(*
---Get axis errir txt
*)
METHOD Get_ErrTxt : STRING(255)
VAR_INPUT
END_VAR
Get_ErrTxt:=fb_motionModule.axisErrTxt;
END_METHOD

(*
---Get axis HOME condition
*)
METHOD Get_HomeCondition : BOOL
VAR_INPUT
END_VAR
Get_HomeCondition:=fb_motionModule.homeCondition;
END_METHOD

(*
---Get axis home state
*)
METHOD Get_HomeState : BOOL
VAR_INPUT
END_VAR
Get_HomeState:=fb_motionModule.axisHomeState;
END_METHOD

(*
---Get axis JOG condition
*)
METHOD Get_JogCondition : BOOL
VAR_INPUT
END_VAR
Get_JogCondition:=fb_motionModule.jogCondition;
END_METHOD

(*
---Get axis Modulo move condition
*)
METHOD Get_ModuloCondition : BOOL
VAR_INPUT
END_VAR
Get_ModuloCondition:=fb_motionModule.moveModuloCondition;
END_METHOD

(*
---Get axis pause state
*)
METHOD Get_Pause : BOOL
VAR_INPUT
END_VAR
Get_Pause:=fb_motionModule.axisPause;
END_METHOD

(*
---Get axis_ref pointer
*)
METHOD Get_pAXIS_REF : POINTER TO AXIS_REF
VAR_INPUT
END_VAR
Get_pAXIS_REF:=fb_motionModule.pAxis;
END_METHOD

(*
---Get axis REL condition
*)
METHOD Get_RelCondition : BOOL
VAR_INPUT
END_VAR
Get_RelCondition:=fb_motionModule.relCondition;
END_METHOD

(*
---Get axis SetPos condition
*)
METHOD Get_SetPosCondition : BOOL
VAR_INPUT
END_VAR
Get_SetPosCondition:=fb_motionModule.setCondition;
END_METHOD

(*
---Get axis VEL condition
*)
METHOD Get_VelCondition : BOOL
VAR_INPUT
END_VAR
Get_VelCondition:=fb_motionModule.velCondition;
END_METHOD

ACTION Obj_Instance:
fb_motionModule(
	axis:=axis,
	PLimitSwitch:= bPLimitSwitch, 
	NLimitSwitch:= bNLimitSwitch, 
	DOGPointSwitch:= bDOGPointSwitch, 
	bP_Pos:=bP_Pos,
	bN_Pos:=bN_Pos,
	torqueAlmValue:=bTorqueAlmValue,
	torqueEN:=bTorqueEN,
	motorType:= eMotorType, 
	moduloMode:= bModuloMode, 
	errorID:= nBaseErrID, 
	nameTXT:= sNameTXT, 
	axisEnable:= TRUE, 
	bE_Stop:= bE_Stop, 
	axisOverride:= , 
	//ctrlMode:= eCtrlMode,
	hmiEN:= hmiEN, 
	powerEnable:= , 
	powerEnable_Positive:= bEnablePositive, 
	powerEnable_Negative:= bEnableNegative, 
	enableSoftLimit:= bEnableSoftLimit, 
	softPLimitPos:= fSoftPLimitPos, 
	softNLimitPos:= fSoftNLimitPos, 
	axisStopFlag:= , 
	resetExecute:= , 
	pauseExecute:= , 
	jogExecute:= , 
	jogConditionOuter:= bJogConditionOuter, 
	jogDirection:= , 
	jogVelocity:= , 
	jogAcceleration:= , 
	jogDeceleration:= , 
	jogJerk:= , 
	stopExecute:= , 
	stopDeceleration:= , 
	stopJerk:= , 
	absExecute:= , 
	absMixedMovement:= , 
	absConditionOuter:= bAbsConditionOuter, 
	absPosition:= , 
	absVelocity:= , 
	absMixedPositionArray:= , 
	absMixedVelocityArray:= , 
	absMixedArrayLength:= , 
	absAcceleration:= , 
	absDeceleration:= , 
	absJerk:= , 
	relExecute:= , 
	relConditionOuter:= bRelConditionOuter, 
	relDistance:= , 
	relVelocity:= , 
	relAcceleration:= , 
	relDeceleration:= , 
	relJerk:= , 
	velExecute:= , 
	velConditionOuter:= bVelConditionOuter, 
	velDirection:= , 
	velVelocity:= , 
	velAcceleration:= , 
	velDeceleration:= , 
	velJerk:= , 
	homeExecute:= , 
	homeConditionOuter:= bHomeConditionOuter, 
	homeDirection:= bHomeDirection, 
	homeMode:= eHomeMode, 
	homeLimitSwitch_To_DOGDistance:= fHomeLimitSwitch_To_DOGDistance, 
	homeOnlyDOGDistance:= fHomeOnlyDOGDistance, 
	homeOnlyDOGMaxDistance:= fHomeOnlyDOGMaxDistance, 
	homePosition:= fHomePosition, 
	homeCheckRange:= fHomeCheckRange, 
	homeVel:= fHomeVel, 
	homeVelSlow:= fHomeVelSlow, 
	setPosExecute:= , 
	setConditionOuter:= bSetConditionOuter, 
	setPosPosition:= , 
	setPosOptions:= , 
	moveModuloExecute:= , 
	moveModuloConditionOuter:= bMoveModuloConditionOuter, 
	moveModuloPosition:= , 
	moveModuloVelocity:= , 
	moveModuloAcceleration:= , 
	moveModuloDeceleration:= , 
	moveModuloJerk:= , 
	moveModuloDirection:= , 
	axisActualPos=> , 
	axisActualVel=> , 
	axisPause=> , 
	axisBusy=> , 
	axisDone=> , 
	axisError=> , 
	axisErrId=> , 
	axisErrTxt=> , 
	axisHomeState=> , 
	pAxis=> , 
	jogCondition=> , 
	absCondition=> , 
	relCondition=> , 
	velCondition=> , 
	homeCondition=> , 
	setCondition=> , 
	moveModuloCondition=> );
END_ACTION

(*
---Set Acceleration\Deceleration\Jerk
*)
METHOD Set_AccDecJerk : BOOL
VAR_INPUT
	acc:LREAL;//target Acceleration
	dec:LREAL;//target Deceleration
	jerk:LREAL;//target Jerk
END_VAR
fb_motionModule.jogAcceleration:=acc;
fb_motionModule.jogDeceleration:=dec;
fb_motionModule.jogJerk:=jerk;

fb_motionModule.stopDeceleration:=dec;
fb_motionModule.stopJerk:=jerk;

fb_motionModule.absAcceleration:=acc;
fb_motionModule.absDeceleration:=dec;
fb_motionModule.absJerk:=jerk;

fb_motionModule.relAcceleration:=acc;
fb_motionModule.relDeceleration:=dec;
fb_motionModule.relJerk:=jerk;

fb_motionModule.velAcceleration:=acc;
fb_motionModule.velDeceleration:=dec;
fb_motionModule.velJerk:=jerk;

fb_motionModule.moveModuloAcceleration:=acc;
fb_motionModule.moveModuloDeceleration:=dec;
fb_motionModule.moveModuloJerk:=jerk;

Set_AccDecJerk:=TRUE;
END_METHOD

(*
---Set axis override
*)
METHOD Set_Override : BOOL
VAR_INPUT
	override:LREAL;//target axis override
END_VAR
fb_motionModule.axisOverride:=override;

Set_Override:=TRUE;
END_METHOD

(*
---Set Power Enable
*)
METHOD Set_Power : BOOL
VAR_INPUT
	enable:BOOL;
END_VAR
fb_motionModule.powerEnable:=enable;
END_METHOD

ACTION VersionLog:
(*
Version: V1.0.0.0
/-----------------------------------------------/
Version: V1.0.0.1
修改：修改电机模块使能触发方式(Add method Set_Power)
/-----------------------------------------------/
Version: V1.0.0.2
修改：增加中文报警输出
/-----------------------------------------------/
Version: V1.0.0.3
修改：增加中优化代码
/-----------------------------------------------/
Version: V1.0.0.4
更新时间: 2020/10/06
修改：配合轴模块更新
/-----------------------------------------------/
*)
END_ACTION

END_FUNCTION_BLOCK

// ---- POUs/BaseModule/ActionModule/motorModule/MotionModule.TcPOU
(*
--报错编号0: 无报错
--报错编号1: E_Stop!!!
--报错编号2: Soft Limit Error
--报错编号3: PLimit Switch Error
--报错编号4: NLimit Switch Error
--报错编号5: Origin sensor cannot be searched
--报错编号6: Go Home Failed
--报错编号7: Absolute Move Error
--报错编号8: JOG Move Error
--报错编号9: Modulo Move Error
--报错编号10: Relative Move Error
--报错编号11: Set Position Error
--报错编号12: Axis Stop Error
--报错编号13: Velocity Move Error
--报错编号14: mcPower Error
--报错编号15: mcReset Error
--报错编号16: axis_Status_Error
*)
FUNCTION_BLOCK MotionModule
VAR_IN_OUT
	axis							:AXIS_REF;//链接到实际的轴
END_VAR
VAR_INPUT
	HMIItf							:motionModuleDataHMI;//for manual and IO control//用于生成一个轴对象手动界面
	PLimitSwitch					:BOOL:=TRUE;//MC轴正限位感应信号
	NLimitSwitch					:BOOL:=TRUE;//MC轴负限位感应信号
	DOGPointSwitch					:BOOL:=FALSE;//MC轴原点感应信号
	bP_Pos							:LREAL:=0.777;	 //正向位置(开门）
	bN_Pos							:LREAL:=0.777;	 //负向位置(关门）

	motorType						:MotorType:=MotorType_Default;//设置电机的类型
	moduloMode						:BOOL:=FALSE;// modulo Mode, 旋转模式
	errorID							:UDINT:=0;//电机错误报警分配的起始ID
	nameTXT							:STRING(255):='';//电机名字

	axisEnable						:BOOL:=TRUE;//轴触摸屏是否启用
	bE_Stop							:BOOL:=TRUE;//急停信号
	axisOverride					:LREAL:=100.0;//轴运动的速度比
	//ctrlMode						:ControlMode:=ControlMode.eManualCtrMode;//eManualCtrMode or eAutoCtrMode
	hmiEN							:BOOL:=TRUE;//HMI 启用条件
	torqueEN						:BOOL:=FALSE;// 启用条件
	torqueAlmValue					:LREAL;// 报警扭力值
//POWER
	powerEnable						:BOOL:=TRUE;//轴使能触发
	powerEnable_Positive			:BOOL:=TRUE;//轴允许正转
	powerEnable_Negative			:BOOL:=TRUE;//轴允许反转
//Soft limit
	enableSoftLimit					:BOOL:=FALSE;//轴软限位 启用信号
	softPLimitPos					:LREAL:=9999999;//轴软限位 正向软限位
	softNLimitPos					:LREAL:=-9999999;//轴软限位 负向软限位
//STOP
	axisStopFlag					:BOOL:=FALSE;//轴是否停止
//RESET
	resetExecute					:BOOL:=TRUE;
	resetExecute2					:BOOL:=TRUE;//轴Reset的触发信号
//PAUSE
	pauseExecute					:BOOL:=FALSE;//轴Pause的触发信号
//JOG
	jogExecute						:BOOL:=FALSE;//轴JOG的触发信号
	jogConditionOuter				:BOOL:=TRUE;//轴JOG运动启停条件Outer
	jogDirection					:BOOL:=TRUE;//轴JOG运动方向信号, TRUE--正向，FALSE--反向
	jogVelocity						:LREAL:=10;//轴JOG运动运行速率值
	jogAcceleration					:LREAL:=0;//轴JOG运动加速度值
	jogDeceleration					:LREAL:=0;//轴JOG运动减速度值
	jogJerk							:LREAL:=0;//轴JOG运动 加加速度
//STOP
	stopExecute						:BOOL:=FALSE;//轴STOP的触发信号
	//20211029新增---by CPH 目的是仅有原点信号进行回零时，Stopexcute或者ACT——Stop动作无法似的该轴停止
	stoptemp						:BOOL:=FALSE;//轴STOP中转变量，主要传递给HMI界面的Stop指令
	stopDeceleration				:LREAL:=0;//轴STOP运动减速度值
	stopJerk						:LREAL:=0;//轴STOP运动 加加速度
//MoveAbsolute
	absExecute						:BOOL:=FALSE;//轴绝对运动的启停信号
	absMixedMovement				:BOOL:=FALSE;//轴绝对运动的混合变速运动 启用
	absConditionOuter				:BOOL:=TRUE;//轴绝对运动启停条件Outer
	absPosition						:LREAL:=0;//轴绝对运动 目标位置
	absVelocity						:LREAL:=0; //轴绝对运动 运行速率值
	absMixedPositionArray			:ARRAY [1..50] OF LREAL;//轴绝对运动 混合目标位置 变速触发位置数组 最大50个 数组最后一个位置为终点目标位置
	absMixedVelocityArray			:ARRAY [1..50] OF LREAL;//轴绝对运动 混合目标位置 变速触发位置数组 最大50个
	absMixedArrayLength				:UDINT:=0;//轴绝对运动 混合变速触发位置数组 长度 最大50个
	absAcceleration					:LREAL:=0;//轴绝对运动 加速度值
	absDeceleration					:LREAL:=0;//轴绝对运动 减速度值
	absJerk							:LREAL:=0;//轴绝对运动 加加速度
//Relative
	relExecute						:BOOL:=FALSE;//轴相对运动的启停信号
	relConditionOuter				:BOOL:=TRUE;//轴相对运动启停条件Outer
	relDistance						:LREAL:=0; //轴相对运动目标位置
	relVelocity						:LREAL:=0; //轴相对运动运行速率值
	relAcceleration					:LREAL:=0;//轴相对运动加速度值
	relDeceleration					:LREAL:=0;//轴相对运动减速度值
	relJerk							:LREAL:=0;//轴相对运动 加加速度
//Velocity
	velExecute						:BOOL:=FALSE;//轴速度模式运动的启停信号
	velConditionOuter				:BOOL:=TRUE;//轴速度模式启停条件Outer
	velDirection					:BOOL:=TRUE;//方向信号，TRUE--MC_Positive_Direction, FALSE--MC_Negative_Direction
	velVelocity						:LREAL:=10; //轴速度模式运行速率值
	velAcceleration					:LREAL:=0;//轴速度模式加速度值
	velDeceleration					:LREAL:=0;//轴速度模式减速度值
	velJerk							:LREAL:=0;//轴速度模式 加加速度
//Home
	homeExecute						:BOOL:=FALSE;//轴go home的启停信号
	homeConditionOuter				:BOOL:=TRUE;//轴go home的启停条件Outer
	homeDirection					:BOOL:=TRUE;//轴go home方向 TRUE--正方向，FALSE--负方向
	homeMode						:MotorHomeMode:=MotorHomeMode.MotorHomeMode_Default;//轴go home 模式
	homeLimitSwitch_To_DOGDistance	:LREAL:=5;//电机Home模式为 MotorHomeMode_PLimitSwitch_To_DOG/MotorHomeMode_NLimitSwitch_To_DOG 时, 脱离限位为原点的距离值
	homeOnlyDOGDistance				:LREAL:=5;//电机Home模式为 MotorHomeMode_OnlyDOGPointSwitch 时, 执行往复搜寻动作的幅度
	homeOnlyDOGMaxDistance			:LREAL:=360;//电机Home模式为 MotorHomeMode_OnlyDOGPointSwitch 时, 执行往复搜寻动作幅度的最大值
	homePosition					:LREAL:=0;
	homeCheckRange					:LREAL:=0.01;//轴go home执行完后当前位置判断值
	homeVel							:LREAL:=10;//轴go home 查找限位的速率
	homeVelSlow						:LREAL:=5;//轴go home 查找限位的爬行速率
//SetPositon
	setPosExecute					:BOOL:=FALSE;//轴当前位置设定启停信号
	setConditionOuter				:BOOL:=TRUE;//轴当前位置设定启停条件Outer
	setPosPosition					:LREAL:=0; //轴当前位置设定值
	setPosOptions					:ST_SetPositionOptions;//:=ST_SetPositionOptions.ClearPositionLag;
//MC_MoveModulo
	moveModuloExecute				:BOOL:=FALSE;//轴模运动的启停信号
	moveModuloConditionOuter		:BOOL:=TRUE;//轴模运动启停条件Outer
	moveModuloPosition				:LREAL:=0;//轴模运动目标位置
	moveModuloVelocity				:LREAL:=100; //轴模运动运行速率值
	moveModuloAcceleration			:LREAL:=0;//轴模运动加速度值
	moveModuloDeceleration			:LREAL:=0;//轴模运动减速度值
	moveModuloJerk					:LREAL:=0;//轴模运动 加加速度
	moveModuloDirection				:MC_Direction:=MC_Direction.MC_Shortest_Way;//MC_Shortest_Way; MC_Positive_Direction; MC_Negative_Direction
	noteWTXT_jog					:WSTRING(255):="";// 轴点动动作NoteTXT 中文
	noteWTXT_abs					:WSTRING(255):="";// 轴绝对定位动作NoteTXT 中文
	noteWTXT_rel					:WSTRING(255):="";// 轴相对定位动作NoteTXT 中文
	noteWTXT_vel					:WSTRING(255):="";// 轴速度运动动作NoteTXT 中文
END_VAR
VAR_OUTPUT
	axisActualPos					:LREAL:=0;//轴的实际位置
	axisActualVel					:LREAL:=0;//轴的实际速率
	axisActualtorque				:LREAL:=0;//轴的实际扭力
	axisPause						:BOOL;//轴的Pause状态
	axisBusy						:BOOL;//轴的Busy状态
	axisDone						:BOOL;//轴的Done状态
	axisError						:BOOL;//轴的Error状态
	axisErrId						:UDINT;//轴的Error Id值
	axisErrTxt						:STRING(255);//轴的报错文本信息
	axisErrWTxt						:WSTRING(255);//轴的报错文本信息 中文
	axisHomeState					:BOOL:=FALSE;//轴的原点状态
	pAxis	  						:POINTER TO AXIS_REF;
	
	note_jog						:BOOL:=FALSE;// 点动条件不满足
	jogCondition					:BOOL;//轴JOG运动启动条件
	note_abs						:BOOL:=FALSE;// 绝对定位条件不满足
	absCondition					:BOOL;//轴绝对运动启动条件
	note_rel						:BOOL:=FALSE;// 相对定位条件不满足
	relCondition					:BOOL;//轴相对运动启动条件
	note_vel						:BOOL:=FALSE;// 速度条件不满足
	velCondition					:BOOL;//轴速度模式启动条件
	note_home						:BOOL:=FALSE;// 回原条件不满足
	homeCondition					:BOOL;//轴go home的启动条件
	setCondition					:BOOL;//轴当前位置设定启动条件
	moveModuloCondition				:BOOL;//轴模运动启动条件
END_VAR
VAR
	//axis							:AXIS_REF;//链接到实际的轴

	op_mode 				AT%Q*	:SINT:=8;//RxPDO1的Modes of operation---只用于横川DD马达(高创驱动器)
	mode_display 			AT%I*	:SINT;//TxPDO1的Modes of operation display---只用于横川DD马达(高创驱动器)
	maxProfileVelocity  	AT%Q*	:UDINT:=838860800 ; //链接到伺服的Maxprofilevelocity
	statusWord 				AT%I*	:UINT; //链接到伺服的Statusword
	
	torqueAlmErr					:BOOL;// 报警扭力
	torqueErr_Rtrig					:R_TRIG;
	bInit							:BOOL:=FALSE;
	mcBusy							:BOOL;
	mcError							:BOOL;
	mcPower							:MC_Power;
	mcReset							:MC_Reset;
	mcStop							:MC_Stop;
//	mcHalt							:MC_Halt;
	mcJog							:MC_Jog;
	mcABSMove						:MC_MoveAbsolute;
	mcABSMove2						:MC_MoveAbsolute;
	mcABSMove3						:MC_MoveAbsolute;
	mcABSMove4						:MC_MoveAbsolute;
	absBufferMode					:MC_BufferMode:=MC_BufferMode.MC_Aborting;
	mcRel							:MC_MoveRelative;
	mcVel							:MC_MoveVelocity;
	mcHome							:MC_Home;
	mcSetPos						:MC_SetPosition;
	mcMoveModulo					:MC_MoveModulo;
//STOP
	stopBusy						:BOOL;
	stopDone						:BOOL;
	stopErrorDone					:BOOL;
	stopTrigR1						:R_Trig;//上升沿触发
	stopStep						:UINT:=0;
	stopTimeout						:TON;
//Jog
	jogBusy							:BOOL;
	jogDone							:BOOL;
	jogErrorDone					:BOOL;
	jogForward						:BOOL:=FALSE;//轴JOG运动正向启停信号
	jogBackwards					:BOOL:=FALSE;//轴JOG运动反向启停信号
	jogTrigR1						:R_Trig;//上升沿触发
	jogTrigF1						:F_Trig;//上升沿触发
	jogTrigR1_NAiko					:R_Trig;//上升沿触发
	jogTrigF1_NAiko					:F_Trig;//上升沿触发
	jogTrigR1_PAiko					:R_Trig;//上升沿触发
	jogTrigF1_PAiko					:F_Trig;//上升沿触发
	
	jogStep							:UINT:=0;
//Absolute
	absBusy							:BOOL;
	absDone							:BOOL;
	absErrorDone					:BOOL;
	absTrigR1						:R_Trig;//上升沿触发
	absT1							:TON;//长按计时
	absRP							:R_TRIG;// 短按执行去开门位置
	absRN							:R_TRIG;// 短按执行去关门位置
	absStep							:UINT:=0;
	absMixedCount					:UDINT:=0;
//Relative
	relBusy							:BOOL;
	relDone							:BOOL;
	relErrorDone					:BOOL;
	relTrigR1						:R_Trig;//上升沿触发
	relT1							:TON;//长按计时
	relStep							:UINT:=0;
//Velocity 
	velBusy							:BOOL;
	velDone							:BOOL;
	velErrorDone					:BOOL;
	velTrigR1						:R_Trig;//上升沿触发
	velStep							:UINT:=0;
	velChangeVel					:BOOL:=FALSE;//轴速度模式运动 速度改变触发
	
	velTrigR1_NAiko					:R_Trig;//上升沿触发
	velTrigF1_NAiko					:F_Trig;//上升沿触发
	velTrigR1_PAiko					:R_Trig;//上升沿触发
	velTrigF1_PAiko					:F_Trig;//上升沿触发
//Home
	goHomeTrigR1					:R_Trig;//上升沿触发
	goHomeTrigF1					:F_Trig;//下降沿检测
	goHomeDelayTon					:Ton;
	goHomeDelayTime					:TIME:=T#100MS;
	goHomeRelDistance				:LREAL:=0; //Home 轴相对运动目标位置
	goHomeRelVelocity				:LREAL:=0; //Home 轴相对运动运行速率值

	homeDone						:BOOL;
	homeErrorDone					:BOOL;
	homeBusy						:BOOL;
	homeStep						:UINT:=0;
//SetPositon
	setPosBusy						:BOOL;
	setPosDone						:BOOL;
	setPosErrorDone					:BOOL;
	setPosTrigR1					:R_Trig;//上升沿触发
	setPosStep						:UINT:=0;
//MC_MoveModulo
	moveModuloBusy					:BOOL;
	moveModuloDone					:BOOL;
	moveModuloErrorDone				:BOOL;
	moveModuloStep					:UINT:=0;
//power
	powerTrigF1						:F_Trig;//下降沿触发
	powerEnable_Inner				:BOOL:=TRUE;//轴使能触发 内部的
	powerReady						:BOOL;
//reset
	resetBusy						:BOOL;
	resetDone						:BOOL;
	resetErrorDone					:BOOL;
	resetTrigR1						:R_Trig;//上升沿触发
	resetTrigR2						:R_Trig;//上升沿触发
	resetStep						:UINT:=0;
//pause
	pause_Manual_F_Trig				:F_Trig;//HMI暂停 上升沿触发
	pauseR_Trig						:R_Trig;//暂停 上升沿触发
	pauseF_Trig						:F_Trig;//暂停 下降沿触发
//Loop
	loopRelGoTrigR1					:R_Trig;//上升沿触发
	loopAbsGoTrigR1					:R_Trig;//上升沿触发
	loopRelGoT1						:TON;//长按计时
	loopAbsGoT1						:TON;//长按计时
	loopStepHome					:UINT:=0;
	loopStep						:UINT:=0;
	loopRelGo						:BOOL:=FALSE;//loop 相对运动启动
	loopGoHome						:BOOL:=FALSE;//loop 相对运动启动 回原方式
	loopAbsGo						:BOOL:=FALSE;//loop 绝对运动启动
	loopFirstPoint					:LREAL:=0;//loop 第1个点
	loopSecondPoint					:LREAL:=0;//loop 第2个点
	loopGoVel						:LREAL:=10;//loop 运动速率
	loopCycle						:UINT:=0;//loop 循环次数 一次往复才算一次
	loopCycleMax					:UINT:=0;//loop 循环次数 一次往复才算一次
	loopWatingTime					:UINT:=1000;//loop 停留时间（单位ms）
	loopCycleTimes					:UINT:=0;//loop 循环次数 一次往复才算一次
	loopCycleTimesHome				:UINT:=0;//loop 循环次数 一次往复才算一次
	loopWatingTON					:TON;
//Other
	bPLimitSwitch					:BOOL:=TRUE;//MC轴正限位感应信号
	bNLimitSwitch					:BOOL:=TRUE;//MC轴负限位感应信号
	bSoftPLimit						:BOOL:=TRUE;//
	bSoftNLimit						:BOOL:=TRUE;//
	
	overrideSet						:LREAL:=100.0;//轴运动的速度比 设置
	overrideTemp					:LREAL:=100.0;//轴运动的速度比 缓存
	stopTon							:TON;
	manualStep						:UINT:=0;
	busy							:BOOL:=FALSE;
	busyR_Trig						:R_Trig;
	doneR_Trig						:R_Trig;
	motorError						:BOOL:=FALSE;
	PTPErrID						:UDINT;
	errorStep						:UINT:=0;
	
	//OnlyDOG Go home TON
	t1Temp							:TON;
	//Home Delay
	tHomeTemp						:TON;
	loopHomeToPosGoT1				:TON;//长按计时
	loopHomeToPosTrigR1				:R_Trig;//上升沿触发
	noteTON_P:tON;            // 操作提示标志位延时继电器
	noteTON_N:tON;            // 操作提示标志位延时继电器
	noteRTrig_P:R_TRIG;          // 操作提示
	noteRTrig_N:R_TRIG;          // 操作提示
END_VAR

(*
Please refer to the VersionLog file for version records
*)
axis.ReadStatus();
IF moduloMode THEN
	axisActualPos:=axis.NcToPlc.ModuloActPos;//获取轴的实际位置, modulo Mode
ELSE
	axisActualPos:=axis.NcToPlc.ActPos;//获取轴的实际位置
END_IF
axisActualtorque:=axis.NcToPlc.ActTorque;
IF torqueEN THEN// 扭力报警监控
	IF ABS(axisActualtorque)>torqueAlmValue THEN
		torqueAlmErr:=TRUE;
	ELSE
		torqueAlmErr:=FALSE;
	END_IF
ELSE
	torqueAlmErr:=FALSE;
END_IF
torqueErr_Rtrig(CLK:=torqueAlmErr);
IF torqueErr_Rtrig.Q THEN
	errorStep:=17;
END_IF
axisActualVel:=axis.NcToPlc.ActVelo;//获取轴的实际速率
pAxis:=ADR(axis);
powerReady:=mcPower.Status;

IF NOT bE_Stop THEN
	axisStopFlag:=TRUE;
	axisHomeState:=FALSE;
	homeBusy:=FALSE;
	errorStep:=1;
END_IF
bPLimitSwitch:=PLimitSwitch;
bNLimitSwitch:=NLimitSwitch;
bSoftPLimit:=(NOT enableSoftLimit OR ((enableSoftLimit AND axisActualPos<softPLimitPos) OR homeBusy));
bSoftNLimit:=(NOT enableSoftLimit OR ((enableSoftLimit AND axisActualPos>softNLimitPos) OR homeBusy));

busy:=stopBusy OR jogBusy OR absBusy OR relBusy OR velBusy (*OR homeBusy*) OR 0<>loopStep;
mcBusy:=mcStop.Busy OR mcJog.Busy OR mcABSMove.Busy OR mcABSMove2.Busy 
			OR mcABSMove3.Busy OR mcABSMove4.Busy OR mcRel.Busy 
			OR mcVel.Busy OR mcHome.Busy OR mcSetPos.Busy OR mcMoveModulo.Busy;
axisBusy:=(mcBusy OR busy OR homeBusy OR (0<>axis.NcToPlc.AxisState));
busyR_Trig(CLK:=axisBusy);
IF busyR_Trig.Q THEN
	jogDone:=FALSE;
	absDone:=FALSE;
	relDone:=FALSE;
	velDone:=FALSE;
	homeDone:=FALSE;
	setPosDone:=FALSE;
	stopDone:=FALSE;
	moveModuloDone:=FALSE;
	
	axisDone:=FALSE;
END_IF

doneR_Trig(CLK:=(jogDone OR absDone OR relDone OR velDone OR homeDone OR setPosDone (*OR stopDone*) OR moveModuloDone) AND NOT axisBusy);
IF doneR_Trig.Q THEN
	axisDone:=TRUE;
	
	jogDone:=FALSE;
	absDone:=FALSE;
	relDone:=FALSE;
	velDone:=FALSE;
	homeDone:=FALSE;
	setPosDone:=FALSE;
	stopDone:=FALSE;
	moveModuloDone:=FALSE;
END_IF

IF axis.Status.Error OR 0<>axis.NcToPlc.ErrorCode THEN
	errorStep:=16;
END_IF
Error_ACT();
mcError:=mcPower.Error OR mcReset.Error OR mcStop.Error OR mcJog.Error OR mcABSMove.Error 
			OR mcABSMove2.Error OR mcABSMove3.Error OR mcABSMove4.Error 
			 OR mcRel.Error OR mcVel.Error OR mcHome.Error OR mcSetPos.Error
			 OR mcMoveModulo.Error;
axisError:=(mcError OR axis.Status.Error OR 0<>axis.NcToPlc.ErrorCode OR NOT bE_Stop OR motorError OR torqueAlmErr);
Error_ACT();

IF NOT axisError THEN
	errorStep:=0;
END_IF

Power_ACT();
Reset_ACT();
ResetEx_ACT();
SetPause_ACT();
InitHMI_ACT();
ManualCtr_ACT();

Stop_ACT();
JogMove_ACT();
VelMove_ACT();
GoHome_ACT();
RelMove_ACT();
AbsMove_ACT();
MoveModulo_ACT();
SetPosition_ACT();
LoopMove_ACT();
LoopHomeToPos_ACT();
IF NOT bInit THEN
	bInit:=TRUE;
END_IF

busy:=stopBusy OR jogBusy OR absBusy OR relBusy OR velBusy (*OR homeBusy*) OR 0<>loopStep;
mcBusy:=mcStop.Busy OR mcJog.Busy OR mcABSMove.Busy OR mcABSMove2.Busy 
			OR mcABSMove3.Busy OR mcABSMove4.Busy OR mcRel.Busy 
			OR mcVel.Busy OR mcHome.Busy OR mcSetPos.Busy OR mcMoveModulo.Busy;
axisBusy:=(mcBusy OR busy OR homeBusy OR (0<>axis.NcToPlc.AxisState));
busyR_Trig(CLK:=axisBusy);
IF busyR_Trig.Q THEN
	jogDone:=FALSE;
	absDone:=FALSE;
	relDone:=FALSE;
	velDone:=FALSE;
	homeDone:=FALSE;
	setPosDone:=FALSE;
	stopDone:=FALSE;
	moveModuloDone:=FALSE;
	
	axisDone:=FALSE;
END_IF

doneR_Trig(CLK:=(jogDone OR absDone OR relDone OR velDone OR homeDone OR setPosDone (*OR stopDone*) OR moveModuloDone) AND NOT axisBusy);
IF doneR_Trig.Q THEN
	axisDone:=TRUE;
	
	jogDone:=FALSE;
	absDone:=FALSE;
	relDone:=FALSE;
	velDone:=FALSE;
	homeDone:=FALSE;
	setPosDone:=FALSE;
	stopDone:=FALSE;
	moveModuloDone:=FALSE;
END_IF

ACTION AbsMove_ACT:
//轴绝对运动运行控制--absExecute触发条件是复归型
IF NOT bE_Stop THEN
	absStep:=0;
	absExecute:=FALSE;
END_IF
absCondition:=(axisHomeState AND NOT axisError 
				AND NOT axisStopFlag AND (NOT axisBusy OR 0<>loopStep) 
				AND powerReady AND absConditionOuter 
				AND bE_Stop AND NOT axisPause);

mcABSMove(
	Axis:=axis , 
	Execute:= , 
	Position:= , 
	Velocity:= , 
	Acceleration:= , 
	Deceleration:= , 
	Jerk:= , 
	BufferMode:= , 
	Options:= , 
	Done=> , 
	Busy=> , 
	Active=> , 
	CommandAborted=> , 
	Error=> , 
	ErrorID=> );
mcABSMove2(
	Axis:=axis , 
	Execute:= , 
	Position:= , 
	Velocity:= , 
	Acceleration:= , 
	Deceleration:= , 
	Jerk:= , 
	BufferMode:= , 
	Options:= , 
	Done=> , 
	Busy=> , 
	Active=> , 
	CommandAborted=> , 
	Error=> , 
	ErrorID=> );
mcABSMove3(
	Axis:=axis , 
	Execute:= , 
	Position:= , 
	Velocity:= , 
	Acceleration:= , 
	Deceleration:= , 
	Jerk:= , 
	BufferMode:= absBufferMode, 
	Options:= , 
	Done=> , 
	Busy=> , 
	Active=> , 
	CommandAborted=> , 
	Error=> , 
	ErrorID=> );
mcABSMove4(
	Axis:=axis , 
	Execute:= , 
	Position:= , 
	Velocity:= , 
	Acceleration:= , 
	Deceleration:= , 
	Jerk:= , 
	BufferMode:= absBufferMode, 
	Options:= , 
	Done=> , 
	Busy=> , 
	Active=> , 
	CommandAborted=> , 
	Error=> , 
	ErrorID=> );

CASE absStep OF
0:
	absBusy:=FALSE;
	IF absExecute AND (NOT absCondition OR NOT powerEnable_Negative OR NOT powerEnable_Positive OR absVelocity>0.2) THEN
		note_abs:=TRUE;
		note_jog:=FALSE;
		note_vel:=FALSE;
		note_home:=FALSE;
		note_rel:=FALSE;
	END_IF
	IF absExecute AND absCondition THEN
		absBusy:=TRUE;
		absDone:=FALSE;
		absErrorDone:=FALSE;
		note_abs:=FALSE;
		note_jog:=FALSE;
		note_vel:=FALSE;
		note_home:=FALSE;
		note_rel:=FALSE;
		IF NOT absMixedMovement THEN
			absStep:=20;//点到点运动
		ELSE
			absPosition:=absMixedPositionArray[absMixedArrayLength];
			absStep:=100;//多段变速运动
		END_IF
	END_IF
	absExecute:=FALSE;
	absMixedMovement:=FALSE;
	absMixedCount:=1;
	mcABSMove(
		Axis:=axis , 
		Execute:=FALSE ,);
	mcABSMove2(
		Axis:=axis , 
		Execute:=FALSE ,);
	mcABSMove3(
		Axis:=axis , 
		Execute:=FALSE ,);
	mcABSMove4(
		Axis:=axis , 
		Execute:=FALSE ,);
20:
//	正确逻辑
	IF NOT bPLimitSwitch OR NOT bNLimitSwitch OR NOT bSoftPLimit OR NOT bSoftNLimit OR NOT powerEnable_Positive OR NOT powerEnable_Negative THEN
		axisStopFlag:=TRUE;

		IF NOT bPLimitSwitch THEN
			errorStep:=3;
		ELSIF NOT bNLimitSwitch THEN
			errorStep:=4;
		END_IF
		IF NOT bSoftPLimit OR NOT bSoftNLimit THEN
			errorStep:=2;
		END_IF
		IF NOT powerEnable_Positive OR NOT powerEnable_Negative THEN
			errorStep:=19;
		END_IF
		absStep:=10000;//error
		RETURN;
	END_IF
//	测试逻辑
//	IF NOT bSoftPLimit OR NOT bSoftNLimit THEN
//		axisStopFlag:=TRUE;

//		IF NOT bSoftPLimit OR NOT bSoftNLimit THEN
//			errorStep:=2;
//		END_IF
//		absStep:=10000;//error
//		RETURN;
//	END_IF
//	IF NOT bPLimitSwitch OR NOT bNLimitSwitch THEN
//		IF NOT bPLimitSwitch AND ABS(axisActualPos-absPosition)>6 THEN
//			axisStopFlag:=TRUE;
//			errorStep:=3;
//			absStep:=10000;//error
//			RETURN;
//		ELSIF NOT bNLimitSwitch AND ABS(axisActualPos-absPosition)>6 THEN
//			axisStopFlag:=TRUE;
//			errorStep:=4;
//			absStep:=10000;//error
//			RETURN;
//		END_IF
//	END_IF
	mcABSMove(
		Axis:=axis , 
		Execute:=TRUE , 
		Position:=absPosition , 
		Velocity:=absVelocity , 
		Acceleration:=absAcceleration , 
		Deceleration:=absDeceleration , 
		Jerk:=absJerk , 
		BufferMode:= , 
		Options:= , 
		Done=> , 
		Busy=> , 
		Active=> , 
		CommandAborted=> , 
		Error=> , 
		ErrorID=> );
// 正常
	IF mcABSMove.Done THEN//mcABSMove.Done信号只保持一个扫描周期
		absStep:=5000;//done
	ELSIF mcABSMove.Error OR mcABSMove.ErrorID<>0 THEN
		errorStep:=7;
		absStep:=10000;//error
	END_IF
// 测试逻辑
//	IF mcABSMove.Done THEN//mcABSMove.Done信号只保持一个扫描周期
//		IF NOT bSoftPLimit OR NOT bSoftNLimit THEN
//			absStep:=5000;//done
//		ELSE
//			errorStep:=7;
//			absStep:=10000;//error
//		END_IF
//	ELSIF mcABSMove.Error OR mcABSMove.ErrorID<>0 THEN
//		errorStep:=7;
//		absStep:=10000;//error
//	END_IF

	IF axisStopFlag OR NOT powerReady OR 0<>stopStep THEN
		absStep:=4000;//stop
	END_IF

//变速运动
100:
	IF NOT bPLimitSwitch OR NOT bNLimitSwitch OR NOT bSoftPLimit OR NOT bSoftNLimit OR NOT powerEnable_Positive OR NOT powerEnable_Negative THEN
		axisStopFlag:=TRUE;

		IF NOT bPLimitSwitch THEN
			errorStep:=3;
		ELSIF NOT bNLimitSwitch THEN
			errorStep:=4;
		END_IF
		IF NOT bSoftPLimit OR NOT bSoftNLimit THEN
			errorStep:=2;
		END_IF
		IF NOT powerEnable_Positive OR NOT powerEnable_Negative THEN
			errorStep:=19;
		END_IF
		absStep:=10000;//error
		RETURN;
	END_IF
	mcABSMove2(
		Axis:=axis , 
		Execute:=TRUE , 
		Position:=absMixedPositionArray[absMixedCount] , 
		Velocity:=absMixedVelocityArray[absMixedCount] , 
		Acceleration:=absAcceleration , 
		Deceleration:=absDeceleration , 
		Jerk:=absJerk , 
		BufferMode:= , 
		Options:= , 
		Done=> , 
		Busy=> , 
		Active=> , 
		CommandAborted=> , 
		Error=> , 
		ErrorID=> );
	
	IF mcABSMove2.Busy AND (absMixedCount<absMixedArrayLength) THEN
		mcABSMove3(
			Axis:=axis , 
			Execute:=FALSE ,);
		IF absMixedVelocityArray[absMixedCount]>absMixedVelocityArray[absMixedCount+1] THEN
			absBufferMode:=MC_BufferMode.MC_BlendingNext;
		ELSE
			absBufferMode:=MC_BufferMode.MC_BlendingPrevious;
		END_IF
		absMixedCount:=absMixedCount+1;
		absStep:=110;
	END_IF
	IF mcABSMove2.Done THEN//mcABSMove.Done信号只保持一个扫描周期
		absStep:=5000;//done
	ELSIF mcABSMove2.Error OR mcABSMove2.ErrorID<>0 THEN
		errorStep:=7;
		absStep:=10000;//error
	END_IF

	IF axisStopFlag OR NOT powerReady OR 0<>stopStep THEN
		absStep:=4000;//stop
	END_IF
110:
	IF NOT bPLimitSwitch OR NOT bNLimitSwitch OR NOT bSoftPLimit OR NOT bSoftNLimit OR NOT powerEnable_Positive OR NOT powerEnable_Negative THEN
		axisStopFlag:=TRUE;

		IF NOT bPLimitSwitch THEN
			errorStep:=3;
		ELSIF NOT bNLimitSwitch THEN
			errorStep:=4;
		END_IF
		IF NOT bSoftPLimit OR NOT bSoftNLimit THEN
			errorStep:=2;
		END_IF
		IF NOT powerEnable_Positive OR NOT powerEnable_Negative THEN
			errorStep:=19;
		END_IF
		absStep:=10000;//error
		RETURN;
	END_IF
	mcABSMove3(
		Axis:=axis , 
		Execute:=TRUE , 
		Position:=absMixedPositionArray[absMixedCount] , 
		Velocity:=absMixedVelocityArray[absMixedCount] , 
		Acceleration:=absAcceleration , 
		Deceleration:=absDeceleration , 
		Jerk:=absJerk , 
		BufferMode:= , 
		Options:= , 
		Done=> , 
		Busy=> , 
		Active=> , 
		CommandAborted=> , 
		Error=> , 
		ErrorID=> );
	
	IF mcABSMove3.Busy AND NOT mcABSMove2.Busy AND NOT mcABSMove4.Busy AND (absMixedCount<absMixedArrayLength) THEN
		mcABSMove4(
			Axis:=axis , 
			Execute:=FALSE ,);
		IF absMixedVelocityArray[absMixedCount]>absMixedVelocityArray[absMixedCount+1] THEN
			absBufferMode:=MC_BufferMode.MC_BlendingNext;
		ELSE
			absBufferMode:=MC_BufferMode.MC_BlendingPrevious;
		END_IF
		absMixedCount:=absMixedCount+1;
		absStep:=120;
	END_IF
	IF mcABSMove3.Done THEN//mcABSMove.Done信号只保持一个扫描周期
		absStep:=5000;//done
	ELSIF mcABSMove3.Error OR mcABSMove3.ErrorID<>0 THEN
		errorStep:=7;
		absStep:=10000;//error
	END_IF

	IF axisStopFlag OR NOT powerReady OR 0<>stopStep THEN
		absStep:=4000;//stop
	END_IF
120:
	IF NOT bPLimitSwitch OR NOT bNLimitSwitch OR NOT bSoftPLimit OR NOT bSoftNLimit OR NOT powerEnable_Positive OR NOT powerEnable_Negative THEN
		axisStopFlag:=TRUE;

		IF NOT bPLimitSwitch THEN
			errorStep:=3;
		ELSIF NOT bNLimitSwitch THEN
			errorStep:=4;
		END_IF
		IF NOT bSoftPLimit OR NOT bSoftNLimit THEN
			errorStep:=2;
		END_IF
		IF NOT powerEnable_Positive OR NOT powerEnable_Negative THEN
			errorStep:=19;
		END_IF
		absStep:=10000;//error
		RETURN;
	END_IF
	mcABSMove4(
		Axis:=axis , 
		Execute:=TRUE , 
		Position:=absMixedPositionArray[absMixedCount] , 
		Velocity:=absMixedVelocityArray[absMixedCount] , 
		Acceleration:=absAcceleration , 
		Deceleration:=absDeceleration , 
		Jerk:=absJerk , 
		BufferMode:= , 
		Options:= , 
		Done=> , 
		Busy=> , 
		Active=> , 
		CommandAborted=> , 
		Error=> , 
		ErrorID=> );
	
	IF mcABSMove4.Busy AND NOT mcABSMove3.Busy AND (absMixedCount<absMixedArrayLength) THEN
		mcABSMove3(
			Axis:=axis , 
			Execute:=FALSE ,);
		IF absMixedVelocityArray[absMixedCount]>absMixedVelocityArray[absMixedCount+1] THEN
			absBufferMode:=MC_BufferMode.MC_BlendingNext;
		ELSE
			absBufferMode:=MC_BufferMode.MC_BlendingPrevious;
		END_IF
		absMixedCount:=absMixedCount+1;
		absStep:=110;
	END_IF
	IF mcABSMove4.Done THEN//mcABSMove.Done信号只保持一个扫描周期
		absStep:=5000;//done
	ELSIF mcABSMove4.Error OR mcABSMove4.ErrorID<>0 THEN
		errorStep:=7;
		absStep:=10000;//error
	END_IF

	IF axisStopFlag OR NOT powerReady OR 0<>stopStep THEN
		absStep:=4000;//stop
	END_IF
	
4000://Stop
	mcABSMove(
		Axis:=axis , 
		Execute:=FALSE ,);
	mcABSMove2(
		Axis:=axis , 
		Execute:=FALSE ,);
	mcABSMove3(
		Axis:=axis , 
		Execute:=FALSE ,);
	mcABSMove4(
		Axis:=axis , 
		Execute:=FALSE ,);
	absExecute:=FALSE;
	absBusy:=FALSE;
	absDone:=FALSE;
	absErrorDone:=FALSE;
	absStep:=0;
5000://Done
	mcABSMove(
		Axis:=axis , 
		Execute:=FALSE ,);
	mcABSMove2(
		Axis:=axis , 
		Execute:=FALSE ,);
	mcABSMove3(
		Axis:=axis , 
		Execute:=FALSE ,);
	mcABSMove4(
		Axis:=axis , 
		Execute:=FALSE ,);
	absExecute:=FALSE;
	absBusy:=FALSE;
	absDone:=TRUE;
	absErrorDone:=FALSE;
	absStep:=0;
10000://Error
	mcABSMove(
		Axis:=axis , 
		Execute:=FALSE ,);
	mcABSMove2(
		Axis:=axis , 
		Execute:=FALSE ,);
	mcABSMove3(
		Axis:=axis , 
		Execute:=FALSE ,);
	mcABSMove4(
		Axis:=axis , 
		Execute:=FALSE ,);
	absExecute:=FALSE;
	absBusy:=FALSE;
	absDone:=FALSE;
	absErrorDone:=TRUE;
	absStep:=0;
END_CASE
END_ACTION

//设定速度运行模式的方向和速度
METHOD changeVelVel
VAR_INPUT
	vel:LREAL;//速度设定
END_VAR
velChangeVel:=TRUE;
velVelocity:=vel;
END_METHOD

ACTION Error_ACT:
CASE errorStep OF
	0:
		motorError:=FALSE;
		axisErrId:=0;
		axisErrTxt:='';
		axisErrWTxt:="";
		PTPErrID:=0;
 (*
	1:
		motorError:=TRUE;
		axisErrId:=errorID+errorStep;
		axisErrTxt:=CONCAT(STR1:=nameTXT,STR2:=' E_Stop!!!');
		axisErrWTxt:=WCONCAT(STR1:=TO_WSTRING(nameTXT),STR2:=" 急停错误!!!");
	2:
		motorError:=TRUE;
		axisErrId:=errorID+errorStep;
		axisErrTxt:=CONCAT(STR1:=nameTXT,STR2:=' Soft Limit Error');
		axisErrWTxt:=WCONCAT(STR1:=TO_WSTRING(nameTXT),STR2:=" 软限位错误");
	3:
		motorError:=TRUE;
		axisErrId:=errorID+errorStep;
		axisErrTxt:=CONCAT(STR1:=nameTXT,STR2:=' PLimit Switch Error');
		axisErrWTxt:=WCONCAT(STR1:=TO_WSTRING(nameTXT),STR2:=" 正限位感应错误");
	4:
		motorError:=TRUE;
		axisErrId:=errorID+errorStep;
		axisErrTxt:=CONCAT(STR1:=nameTXT,STR2:=' NLimit Switch Error');
		axisErrWTxt:=WCONCAT(STR1:=TO_WSTRING(nameTXT),STR2:=" 负限位感应错误");
	5:
		motorError:=TRUE;
		axisErrId:=errorID+errorStep;
		axisErrTxt:=CONCAT(STR1:=nameTXT,STR2:=' Origin sensor cannot be searched');
		axisErrWTxt:=WCONCAT(STR1:=TO_WSTRING(nameTXT),STR2:=" 原点信号无法被搜索到");
	6:
		motorError:=TRUE;
		axisErrId:=errorID+errorStep;
		axisErrTxt:=CONCAT(STR1:=nameTXT,STR2:=' Go Home Failed');
		axisErrWTxt:=WCONCAT(STR1:=TO_WSTRING(nameTXT),STR2:=" 回原点失败");
	7:
		motorError:=TRUE;
		axisErrId:=errorID+errorStep;
		axisErrTxt:=CONCAT(STR1:=nameTXT,STR2:=' Absolute Move Error');
		axisErrWTxt:=WCONCAT(STR1:=TO_WSTRING(nameTXT),STR2:=" 绝对定位错误");
	8:
		motorError:=TRUE;
		axisErrId:=errorID+errorStep;
		axisErrTxt:=CONCAT(STR1:=nameTXT,STR2:=' JOG Move Error');
		axisErrWTxt:=WCONCAT(STR1:=TO_WSTRING(nameTXT),STR2:=" JOG运动错误");
	9:
		motorError:=TRUE;
		axisErrId:=errorID+errorStep;
		axisErrTxt:=CONCAT(STR1:=nameTXT,STR2:=' Modulo Move Error');
		axisErrWTxt:=WCONCAT(STR1:=TO_WSTRING(nameTXT),STR2:=" 模值定位错误");
	10:
		motorError:=TRUE;
		axisErrId:=errorID+errorStep;
		axisErrTxt:=CONCAT(STR1:=nameTXT,STR2:=' Relative Move Error');
		axisErrWTxt:=WCONCAT(STR1:=TO_WSTRING(nameTXT),STR2:=" 相对定位错误");
	11:
		motorError:=TRUE;
		axisErrId:=errorID+errorStep;
		axisErrTxt:=CONCAT(STR1:=nameTXT,STR2:=' Set Position Error');
		axisErrWTxt:=WCONCAT(STR1:=TO_WSTRING(nameTXT),STR2:=" 设置位置错误");
	12:
		motorError:=TRUE;
		axisErrId:=errorID+errorStep;
		axisErrTxt:=CONCAT(STR1:=nameTXT,STR2:=' Axis Stop Error');
		axisErrWTxt:=WCONCAT(STR1:=TO_WSTRING(nameTXT),STR2:=" 轴停止错误");
	13:
		motorError:=TRUE;
		axisErrId:=errorID+errorStep;
		axisErrTxt:=CONCAT(STR1:=nameTXT,STR2:=' Velocity Move Error');
		axisErrWTxt:=WCONCAT(STR1:=TO_WSTRING(nameTXT),STR2:=" 速度运行错误");
	14:
		motorError:=TRUE;
		axisErrId:=errorID+errorStep;
		axisErrTxt:=CONCAT(STR1:=nameTXT,STR2:=' mcPower Error');
		axisErrWTxt:=WCONCAT(STR1:=TO_WSTRING(nameTXT),STR2:=" mcPower轴使能错误");
	15:
		motorError:=TRUE;
		axisErrId:=errorID+errorStep;
		axisErrTxt:=CONCAT(STR1:=nameTXT,STR2:=' mcReset Error');
		axisErrWTxt:=WCONCAT(STR1:=TO_WSTRING(nameTXT),STR2:=" mcReset轴复位错误");
	16:
		motorError:=TRUE;
		axisErrId:=errorID+errorStep;
		axisErrTxt:=CONCAT(STR1:=nameTXT,STR2:=' axis_Status_Error');
		axisErrWTxt:=WCONCAT(STR1:=TO_WSTRING(nameTXT),STR2:=" 轴状态错误");
 *)
	1..19:
		motorError:=TRUE;
		axisErrId:=getErrID(errorStep);
		axisErrTxt:=getErrTXT(errorStep);
		axisErrWTxt:=getErrWTXT(errorStep);
END_CASE
IF mcPower.Error THEN
	PTPErrID:=mcPower.ErrorID;
END_IF
IF mcReset.Error THEN
	PTPErrID:=mcReset.ErrorID;
END_IF
IF mcStop.Error THEN
	PTPErrID:=mcStop.ErrorID;
END_IF
IF mcJog.Error THEN
	PTPErrID:=mcJog.ErrorID;
END_IF
IF mcABSMove.Error THEN
	PTPErrID:=mcABSMove.ErrorID;
END_IF
IF mcABSMove2.Error THEN
	PTPErrID:=mcABSMove2.ErrorID;
END_IF
IF mcABSMove3.Error THEN
	PTPErrID:=mcABSMove3.ErrorID;
END_IF
IF mcABSMove4.Error THEN
	PTPErrID:=mcABSMove4.ErrorID;
END_IF
IF mcRel.Error THEN
	PTPErrID:=mcRel.ErrorID;
END_IF
IF mcVel.Error THEN
	PTPErrID:=mcVel.ErrorID;
END_IF
IF mcHome.Error THEN
	PTPErrID:=mcHome.ErrorID;
END_IF
IF mcSetPos.Error THEN
	PTPErrID:=mcSetPos.ErrorID;
END_IF
IF mcMoveModulo.Error THEN
	PTPErrID:=mcMoveModulo.ErrorID;
END_IF
IF axis.Status.Error THEN
	PTPErrID:=axis.Status.ErrorID;
END_IF
IF 0<>axis.NcToPlc.ErrorCode THEN
	PTPErrID:=axis.NcToPlc.ErrorCode;
END_IF
END_ACTION

METHOD getErrID : UDINT
VAR_INPUT
	errID					:UDINT;//取值范围1~16
END_VAR
VAR
	nErrID					:UDINT;
END_VAR
nErrID:=errorID+errID;

getErrID:=nErrID;
END_METHOD

METHOD getErrTXT : STRING(255)
VAR_INPUT
	errID					:UDINT;//取值范围1~16
END_VAR
VAR
	sErrTXT					:STRING(255);
END_VAR

CASE errID OF
	1:
		sErrTXT:=CONCAT(STR1:=nameTXT,STR2:=' E_Stop!!!');
	2:
		sErrTXT:=CONCAT(STR1:=nameTXT,STR2:=' Soft Limit Error');
	3:
		sErrTXT:=CONCAT(STR1:=nameTXT,STR2:=' PLimit Switch Error');
	4:
		sErrTXT:=CONCAT(STR1:=nameTXT,STR2:=' NLimit Switch Error');
	5:
		sErrTXT:=CONCAT(STR1:=nameTXT,STR2:=' Origin sensor cannot be searched');
	6:
		sErrTXT:=CONCAT(STR1:=nameTXT,STR2:=' Go Home Failed');
	7:
		sErrTXT:=CONCAT(STR1:=nameTXT,STR2:=' Absolute Move Error');
	8:
		sErrTXT:=CONCAT(STR1:=nameTXT,STR2:=' JOG Move Error');
	9:
		sErrTXT:=CONCAT(STR1:=nameTXT,STR2:=' Modulo Move Error');
	10:
		sErrTXT:=CONCAT(STR1:=nameTXT,STR2:=' Relative Move Error');
	11:
		sErrTXT:=CONCAT(STR1:=nameTXT,STR2:=' Set Position Error');
	12:
		sErrTXT:=CONCAT(STR1:=nameTXT,STR2:=' Axis Stop Error');
	13:
		sErrTXT:=CONCAT(STR1:=nameTXT,STR2:=' Velocity Move Error');
	14:
		sErrTXT:=CONCAT(STR1:=nameTXT,STR2:=' mcPower Error');
	15:
		sErrTXT:=CONCAT(STR1:=nameTXT,STR2:=' mcReset Error');
	16:
		sErrTXT:=CONCAT(STR1:=nameTXT,STR2:=' axis_Status_Error');
	17:
		sErrTXT:=CONCAT(STR1:=nameTXT,STR2:=' axis_Torque_Error');
	18:
		sErrTXT:=CONCAT(STR1:=nameTXT,STR2:=' axis_Done_NotSensor');
	19:
		sErrTXT:=CONCAT(STR1:=nameTXT,STR2:=' axis_Negative Or Postive Error');
ELSE
	sErrTXT:=CONCAT(STR1:=nameTXT,STR2:='Null');
END_CASE
getErrTXT:=sErrTXT;
END_METHOD

METHOD getErrWTXT : WSTRING(255)
VAR_INPUT
	errID					:UDINT;//取值范围1~16
END_VAR
VAR
	sErrTXT					:WSTRING(255);
END_VAR

CASE errID OF
	1:
		sErrTXT:=WCONCAT(STR1:=TO_WSTRING(nameTXT),STR2:=" 急停错误!!!");
	2:
		sErrTXT:=WCONCAT(STR1:=TO_WSTRING(nameTXT),STR2:=" 软限位错误");
	3:
		sErrTXT:=WCONCAT(STR1:=TO_WSTRING(nameTXT),STR2:=" 正限位感应错误");
	4:
		sErrTXT:=WCONCAT(STR1:=TO_WSTRING(nameTXT),STR2:=" 负限位感应错误");
	5:
		sErrTXT:=WCONCAT(STR1:=TO_WSTRING(nameTXT),STR2:=" 原点信号无法被搜索到");
	6:
		sErrTXT:=WCONCAT(STR1:=TO_WSTRING(nameTXT),STR2:=" 回原点失败");
	7:
		sErrTXT:=WCONCAT(STR1:=TO_WSTRING(nameTXT),STR2:=" 绝对定位错误");
	8:
		sErrTXT:=WCONCAT(STR1:=TO_WSTRING(nameTXT),STR2:=" JOG运动错误");
	9:
		sErrTXT:=WCONCAT(STR1:=TO_WSTRING(nameTXT),STR2:=" 模值定位错误");
	10:
		sErrTXT:=WCONCAT(STR1:=TO_WSTRING(nameTXT),STR2:=" 相对定位错误");
	11:
		sErrTXT:=WCONCAT(STR1:=TO_WSTRING(nameTXT),STR2:=" 设置位置错误");
	12:
		sErrTXT:=WCONCAT(STR1:=TO_WSTRING(nameTXT),STR2:=" 轴停止错误");
	13:
		sErrTXT:=WCONCAT(STR1:=TO_WSTRING(nameTXT),STR2:=" 速度运行错误");
	14:
		sErrTXT:=WCONCAT(STR1:=TO_WSTRING(nameTXT),STR2:=" mcPower轴使能错误");
	15:
		sErrTXT:=WCONCAT(STR1:=TO_WSTRING(nameTXT),STR2:=" mcReset轴复位错误");
	16:
		sErrTXT:=WCONCAT(STR1:=TO_WSTRING(nameTXT),STR2:=" 轴状态错误");
	17:
		sErrTXT:=WCONCAT(STR1:=TO_WSTRING(nameTXT),STR2:=" 轴扭力超限");
	18:
		sErrTXT:=WCONCAT(STR1:=TO_WSTRING(nameTXT),STR2:=" 轴到位但传感器未感应");
	19:
		sErrTXT:=WCONCAT(STR1:=TO_WSTRING(nameTXT),STR2:=" 轴正向或反向运行条件不满足");
ELSE
	sErrTXT:=WCONCAT(STR1:=TO_WSTRING(nameTXT),STR2:="空");
END_CASE
getErrWTXT:=sErrTXT;
END_METHOD

ACTION GoHome_ACT:
//轴回原点
(*
go home first direction: positive
DOG point side:negative

                  ____
                 |____|  -->
negative |____________|_____________| positive

*)
(*
go home first direction :negative
DOG point side :positive

                       ____
                <--   |____|  
negative |____________|_____________| positive
*)

IF axisStopFlag THEN
	homeStep:=0;
	homeExecute:=FALSE;
	CASE motorType OF
	MotorType_Default:
		;
	MotorType_DDmotor_HC:
		IF 6=mode_display OR 8<>op_mode THEN
			op_mode:=8;
		END_IF
	END_CASE
END_IF
IF NOT bE_Stop THEN
	homeStep:=50000;//Error
	homeExecute:=FALSE;
	CASE motorType OF
	MotorType_Default:
		;
	MotorType_DDmotor_HC:
		IF 6=mode_display OR 8<>op_mode THEN
			op_mode:=8;
		END_IF
	END_CASE
END_IF
homeCondition:=(NOT axisError AND NOT axisBusy 
				AND NOT axisStopFlag AND powerReady 
				AND homeConditionOuter AND bE_Stop AND NOT axisPause);
CASE homeStep OF
	0:
		homeBusy:=FALSE;
		powerEnable_Inner:=TRUE;
		IF homeExecute AND NOT homeCondition THEN
			note_abs:=FALSE;
			note_jog:=FALSE;
			note_vel:=FALSE;
			note_home:=TRUE;
			note_rel:=FALSE;
		END_IF
		IF homeExecute AND homeCondition THEN
			note_abs:=FALSE;
			note_jog:=FALSE;
			note_vel:=FALSE;
			note_home:=FALSE;
			note_rel:=FALSE;
			stopExecute:=TRUE;
			velExecute:=FALSE;
			axisHomeState:=FALSE;
			homeBusy:=TRUE;
			homeDone:=FALSE;
			homeErrorDone:=FALSE;
			CASE motorType OF
			MotorType_Default:
				IF homeMode=MotorHomeMode.MotorHomeMode_Default THEN
					IF homeDirection THEN
						homeStep:=101;	//正方向回原点-增量式
					ELSE
						homeStep:=201;	//负方向回原点-增量式
					END_IF
				ELSIF homeMode=MotorHomeMode.MotorHomeMode_PLimitSwitch_To_DOG THEN
					homeStep:=1000;
				ELSIF homeMode=MotorHomeMode.MotorHomeMode_NLimitSwitch_To_DOG THEN
					homeStep:=2000;
				ELSIF homeMode=MotorHomeMode.MotorHomeMode_OnlyDOGPointSwitch THEN
					homeStep:=3000;
				ELSE
					IF homeDirection THEN
						homeStep:=101;	//正方向回原点-增量式
					ELSE
						homeStep:=201;	//负方向回原点-增量式
					END_IF
				END_IF
			MotorType_DDmotor_HC:
				homeStep:=301;	//横川-绝对零点回归
			MotorType_Absolute:
				homeStep:=401;	//绝对式编码器回归
			END_CASE
		ELSE
			homeBusy:=FALSE;
		END_IF
		mcHome(
				Axis:= axis,
				Execute:= FALSE, 
				HomingMode:= MC_DefaultHoming);//MC_DefaultHoming  MC_Direct
		homeExecute:=FALSE;	
		
(************** 正方向回原点 ********************)
	101://正方向回原点开始
		goHomeDelayTon(in:=(NOT goHomeDelayTon.Q AND 0=stopStep ), PT:=T#500MS);
		IF 0=axis.NcToPlc.AxisState AND NOT busy AND NOT mcBusy AND 0=stopStep AND goHomeDelayTon.Q THEN
			goHomeDelayTon(in:=FALSE);
			homeStep:=homeStep+1;
		END_IF
	102://检测原点or正限位信号
		velVelocity:=HMIItf.goHomeVel;
		velDirection:=TRUE;
		velExecute:=TRUE;
		IF (DOGPointSwitch) OR (NOT bPLimitSwitch) THEN
			homeStep:=homeStep+1;
		END_IF	
	103:
		velExecute:=FALSE;
		IF 0=axis.NcToPlc.AxisState AND NOT busy AND NOT mcBusy THEN
			homeStep:=homeStep+1;
		END_IF
	104:
		velVelocity:=HMIItf.goHomeVel;
		velDirection:=FALSE;
		velExecute:=TRUE;
		homeStep:=homeStep+1;
	105:
		IF NOT bNLimitSwitch THEN
			homeStep:=50000;//Error
			errorStep:=5;
			RETURN;
		END_IF
		goHomeTrigF1(CLK:=(DOGPointSwitch));
		IF goHomeTrigF1.Q THEN
			homeStep:=homeStep+1;
		END_IF
	106:	
		goHomeDelayTon(in:=NOT goHomeDelayTon.Q,PT:=goHomeDelayTime);
		IF goHomeDelayTon.Q THEN
			goHomeDelayTon(in:=FALSE);
			velExecute:=FALSE;
			homeStep:=homeStep+1;
		END_IF
	107:
		IF 0=axis.NcToPlc.AxisState AND NOT busy AND NOT mcBusy THEN
			homeStep:=108;
		END_IF
	108:
		homeStep:=109;
	109:
		IF 0=axis.NcToPlc.AxisState AND NOT busy AND NOT mcBusy THEN
			mcHome(
				Axis:= axis, 
				Execute:= FALSE,  
				HomingMode:= );//MC_DefaultHoming  MC_Direct
			IF NOT mcHome.Busy THEN
				//homeStep:=120;
				homeStep:=110;
			END_IF
		END_IF
	110:
		powerEnable_Inner:=FALSE;
		goHomeDelayTon(in:=NOT goHomeDelayTon.Q,PT:=T#800MS);
		IF goHomeDelayTon.Q AND NOT powerReady THEN
			homeStep:=homeStep+1;
			goHomeDelayTon(in:=FALSE);
		END_IF
	111:
		homeStep:=homeStep+1;
	112:
		powerEnable_Inner:=TRUE;
		goHomeDelayTon(in:=NOT goHomeDelayTon.Q,PT:=T#800MS);
		IF goHomeDelayTon.Q AND powerReady THEN
			homeStep:=homeStep+1;
			goHomeDelayTon(in:=FALSE);
		END_IF
	113:
		homeStep:=homeStep+1;
	114:
		homeStep:=120;
	120:
		mcHome(
				Axis:=axis , 
				Execute:=TRUE , 
				Position:=homePosition , 
				HomingMode:= , //MC_DefaultHoming  MC_Direct
				BufferMode:= , 
				Options:= , 
				bCalibrationCam:= DOGPointSwitch, //DOGPointSwitch
				Done=> , 
				Busy=> , 
				Active=> , 
				CommandAborted=> , 
				Error=> , 
				ErrorID=> );
		IF (*NOT mcHome.Busy*) mcHome.Done AND NOT mcHome.Error THEN
			mcHome(
				Axis:= axis, 
				Execute:= FALSE, 
				HomingMode:= );//MC_DefaultHoming  MC_Direct
			homeStep:=homeStep+1;
		ELSIF mcHome.Error THEN
			homeStep:=160;//Home Error
		END_IF
		
	121:
		goHomeDelayTon(IN:=NOT goHomeDelayTon.Q,PT:=T#500MS);
		IF goHomeDelayTon.Q THEN
			goHomeDelayTon(in:=FALSE);
			homeStep:=homeStep+1;
		END_IF
	122:
		homeStep:=homeStep+1;
		(*mcSetPos(
			Axis:=axis , 
			Execute:=TRUE , 
			Position:=homePosition);
		goHomeDelayTon(in:=NOT goHomeDelayTon.Q,PT:=T#1000MS);//HMIItf.goHomeDelayTime
		IF goHomeDelayTon.Q THEN
			goHomeDelayTon(in:=FALSE);
			homeStep:=homeStep+1;
		END_IF*)
	123:
		IF ABS(axis.NcToPlc.ActPos)<homeCheckRange THEN
			homeStep:=150;
		ELSE
			homeStep:=160;
		END_IF
	
	150://Home Done
		homeStep:=0;
		homeBusy:=FALSE;
		homeDone:=TRUE;
		homeErrorDone:=FALSE;
		axisHomeState:=TRUE;
		
		homeExecute:=FALSE;
		
	160://Home Error
		homeStep:=0;
		homeBusy:=FALSE;
		homeDone:=FALSE;
		homeErrorDone:=TRUE;
		axisHomeState:=FALSE;
		
		homeExecute:=FALSE;
		
		errorStep:=6;
	
(************** 负方向回原点 ********************)
	201://负方向回原点开始
		goHomeDelayTon(in:=(NOT goHomeDelayTon.Q AND 0=stopStep ), PT:=T#500MS);
		IF 0=axis.NcToPlc.AxisState AND NOT busy AND NOT mcBusy AND 0=stopStep AND goHomeDelayTon.Q THEN
			goHomeDelayTon(in:=FALSE);
			homeStep:=homeStep+1;
		END_IF
	202://检测原点or正限位信号
		velVelocity:=HMIItf.goHomeVel;
		velDirection:=FALSE;
		velExecute:=TRUE;
		IF (DOGPointSwitch) OR NOT bNLimitSwitch THEN
			homeStep:=homeStep+1;
		END_IF	
	203:
		velExecute:=FALSE;
		IF 0=axis.NcToPlc.AxisState AND NOT busy AND NOT mcBusy THEN
			homeStep:=homeStep+1;
		END_IF
	204:
		velVelocity:=HMIItf.goHomeVel;
		velDirection:=TRUE;
		velExecute:=TRUE;		
		goHomeTrigF1(CLK:=FALSE);
		homeStep:=homeStep+1;
	205:
		IF NOT bPLimitSwitch THEN
			homeStep:=50000;//Error
			errorStep:=5;
			RETURN;
		END_IF
		goHomeTrigF1(CLK:=DOGPointSwitch);
		IF goHomeTrigF1.Q THEN
			homeStep:=homeStep+1;
		END_IF
	206:	
		goHomeDelayTon(in:=NOT goHomeDelayTon.Q,PT:=goHomeDelayTime);
		IF goHomeDelayTon.Q THEN
			goHomeDelayTon(IN:=FALSE);
			velExecute:=FALSE;
			
			homeStep:=homeStep+1;
		END_IF
	207:
		IF 0=axis.NcToPlc.AxisState AND NOT busy AND NOT mcBusy THEN
			(*velVelocity:=HMIItf.goHomeVelSlow;
			velDirection:=FALSE;
			velExecute:=TRUE;*)
			goHomeTrigF1(CLK:=FALSE);
			homeStep:=homeStep+1;
		END_IF

	208:
		velVelocity:=HMIItf.goHomeVelSlow;
		velDirection:=FALSE;
		velExecute:=TRUE;
		IF NOT bNLimitSwitch THEN//never cover negative limit switch
			homeStep:=50000;//Error
			errorStep:=5;
			RETURN;
		END_IF
	
		goHomeTrigF1(CLK:=DOGPointSwitch);
		IF goHomeTrigF1.Q THEN
			goHomeDelayTon(IN:=FALSE);
			homeStep:=homeStep+1;
		END_IF
	209:
		goHomeDelayTon(in:=NOT goHomeDelayTon.Q,PT:=goHomeDelayTime);
		IF goHomeDelayTon.Q THEN
			velExecute:=FALSE;
			homeStep:=homeStep+1;
		END_IF
	210:
		IF 0=axis.NcToPlc.AxisState AND NOT busy AND NOT mcBusy THEN
			mcHome(
				Axis:= axis, 
				Execute:= FALSE,  
				HomingMode:= );//MC_DefaultHoming  MC_Direct
			IF NOT mcHome.Busy THEN
				//homeStep:=230;
				homeStep:=220;
			END_IF
		END_IF
	220:
		powerEnable_Inner:=FALSE;
		goHomeDelayTon(in:=NOT goHomeDelayTon.Q,PT:=T#800MS);
		IF goHomeDelayTon.Q AND NOT powerReady THEN
			homeStep:=homeStep+1;
			goHomeDelayTon(in:=FALSE);
		END_IF
	221:
		homeStep:=homeStep+1;
	222:
		powerEnable_Inner:=TRUE;
		goHomeDelayTon(in:=NOT goHomeDelayTon.Q,PT:=T#800MS);
		IF goHomeDelayTon.Q AND powerReady THEN
			homeStep:=homeStep+1;
			goHomeDelayTon(in:=FALSE);
		END_IF
	223:
		homeStep:=homeStep+1;
	224:
		homeStep:=230;
		
	230:
		mcHome(
				Axis:=axis , 
				Execute:=TRUE , 
				Position:=homePosition , 
				HomingMode:= , //MC_DefaultHoming  MC_Direct
				BufferMode:= , 
				Options:= , 
				bCalibrationCam:= DOGPointSwitch, 
				Done=> , 
				Busy=> , 
				Active=> , 
				CommandAborted=> , 
				Error=> , 
				ErrorID=> );
		IF (*NOT mcHome.Busy*) mcHome.Done AND NOT mcHome.Error THEN
			mcHome(
				Axis:= axis, 
				Execute:= FALSE, 
				HomingMode:= );//MC_DefaultHoming  MC_Direct
			homeStep:=homeStep+1;
			
		ELSIF mcHome.Error THEN
			homeStep:=260;//Home Error
		END_IF
	231:
		goHomeDelayTon(in:=NOT goHomeDelayTon.Q,PT:=T#500MS);
		IF goHomeDelayTon.Q THEN
			goHomeDelayTon(in:=FALSE);
			homeStep:=homeStep+1;
		END_IF
	232:
		homeStep:=homeStep+1;
		(*mcSetPos(
			Axis:=axis , 
			Execute:=TRUE , 
			Position:=homePosition);
		goHomeDelayTon(in:=NOT goHomeDelayTon.Q,PT:=T#1000MS);//HMIItf.goHomeDelayTime
		IF goHomeDelayTon.Q THEN
			goHomeDelayTon(in:=FALSE);
			homeStep:=homeStep+1;
		END_IF*)
	233:
		IF ABS(axis.NcToPlc.ActPos)<homeCheckRange THEN
			homeStep:=250;
		ELSE
			homeStep:=260;
		END_IF
	
	250://Home Done
		homeStep:=0;
		homeBusy:=FALSE;
		homeDone:=TRUE;
		homeErrorDone:=FALSE;
		axisHomeState:=TRUE;
		
		homeExecute:=FALSE;
	
	260://Home Error
		homeStep:=0;
		homeBusy:=FALSE;
		homeDone:=FALSE;
		homeErrorDone:=TRUE;
		axisHomeState:=FALSE;
		
		homeExecute:=FALSE;
		
		errorStep:=6;
	
(************** 汇川_横川-绝对零点回归 ********************)
	301://汇川_横川-绝对零点回归
		IF 0=axis.NcToPlc.AxisState AND NOT busy THEN
			powerEnable_Inner:=FALSE;
			homeStep:=homeStep+1;
		END_IF
	302:
		IF NOT powerReady THEN
			op_mode:=6;
			homeStep:=homeStep+1;
		END_IF
		goHomeDelayTon(IN:=FALSE);
	303:
		IF 6=mode_display OR 6=op_mode THEN
			powerEnable_Inner:=TRUE;
			goHomeDelayTon(IN:=NOT goHomeDelayTon.Q,PT:=T#100MS);
			IF goHomeDelayTon.Q AND powerReady THEN
				goHomeDelayTon(IN:=FALSE);
				homeStep:=homeStep+1;
			END_IF
		END_IF
	304:
		goHomeDelayTon(IN:=ABS(axis.NcToPlc.ActPos)<homeCheckRange (*AND ABS(axis.NcToPlc.ActVelo)<0.01*)
							AND NOT axis.Status.Error AND 1=statusWord.12 AND 0=statusWord.13,PT:=T#1000MS);
		IF goHomeDelayTon.Q THEN
			goHomeDelayTon(IN:=FALSE);
			homeStep:=homeStep+1;
		ELSIF axis.Status.Error OR 0<>statusWord.13 THEN
			homeStep:=360;//Error
		END_IF
	305:
		goHomeDelayTon(IN:=NOT goHomeDelayTon.Q,PT:=T#10MS);
		IF goHomeDelayTon.Q THEN
			resetExecute:=TRUE;
			goHomeDelayTon(IN:=FALSE);
			homeStep:=homeStep+1;
		END_IF
	306:
		goHomeDelayTon(IN:=NOT goHomeDelayTon.Q,PT:=T#100MS);
		IF NOT mcReset.Busy AND goHomeDelayTon.Q THEN
			homeStep:=homeStep+1;
			goHomeDelayTon(IN:=FALSE);
		END_IF
	307:
		op_mode:=8;
		homeStep:=homeStep+1;
	308:
		IF 8=mode_display OR 8=op_mode THEN
			homeStep:=homeStep+1;
		END_IF
	309:
		goHomeDelayTon(IN:=NOT goHomeDelayTon.Q,PT:=T#100MS);
		IF goHomeDelayTon.Q THEN
			mcSetPos(
				Axis:=axis , 
				Execute:=TRUE , 
				Position:=homePosition);
			homeStep:=homeStep+1;
		END_IF
	310:	
		homeStep:=350;
		
	350://Go Home Done
		homeStep:=0;
		homeBusy:=FALSE;
		homeDone:=TRUE;
		homeErrorDone:=FALSE;
		axisHomeState:=TRUE;
		
		homeExecute:=FALSE;
	
	360://Home Error
		homeStep:=0;
		homeBusy:=FALSE;
		homeDone:=FALSE;
		homeErrorDone:=TRUE;
		axisHomeState:=FALSE;
		
		homeExecute:=FALSE;
		
		errorStep:=6;
		
(************** 绝对式编码器回归 ********************)
	401://绝对式编码器回归
		IF 0=axis.NcToPlc.AxisState AND NOT busy THEN
			homeStep:=homeStep+1;
		END_IF
	402:
		velVelocity:=HMIItf.goHomeVel;
		IF NOT bPLimitSwitch THEN
			velDirection:=FALSE;
			//velExecute:=TRUE;
			homeStep:=403;
		ELSIF NOT bNLimitSwitch THEN
			velDirection:=TRUE;
			//velExecute:=TRUE;
			homeStep:=403;
		ELSE
			homeStep:=405;//结束
		END_IF
		goHomeDelayTon(IN:=FALSE);
	403:
		velExecute:=TRUE;
		homeStep:=404;
	404:
		goHomeDelayTon(IN:=NOT goHomeDelayTon.Q,PT:=T#100MS);
		IF goHomeDelayTon.Q THEN
			IF bPLimitSwitch AND bNLimitSwitch THEN
				homeStep:=405;
			ELSE
				homeStep:=460;
			END_IF
			goHomeDelayTon(IN:=FALSE);
			velExecute:=FALSE;
		END_IF
	405:
		velExecute:=FALSE;
		homeStep:=homeStep+1;
	406:
		IF 0=axis.NcToPlc.AxisState AND NOT busy THEN
			homeStep:=homeStep+1;
		END_IF
	407:
		homeStep:=450;//Home Done
		
	450://Home Done
		homeStep:=0;
		homeBusy:=FALSE;
		homeDone:=TRUE;
		homeErrorDone:=FALSE;
		axisHomeState:=TRUE;
		
		homeExecute:=FALSE;
		
	460://Home Error
		homeStep:=0;
		homeBusy:=FALSE;
		homeDone:=FALSE;
		homeErrorDone:=TRUE;
		axisHomeState:=FALSE;
		
		homeExecute:=FALSE;
		
		errorStep:=6;

(************** 正限位做原点 ********************)
	1000://正方向回原点开始，以正限位做原点
		goHomeDelayTon(in:=(NOT goHomeDelayTon.Q AND 0=stopStep ), PT:=T#500MS);
		IF 0=axis.NcToPlc.AxisState AND NOT busy AND NOT mcBusy AND 0=stopStep AND goHomeDelayTon.Q THEN
			goHomeDelayTon(in:=FALSE);
			homeStep:=homeStep+10;
		END_IF
	1010://正限位信号
		velVelocity:=HMIItf.goHomeVel;
		velDirection:=TRUE;
		velExecute:=TRUE;
		IF (NOT bPLimitSwitch) THEN
			velExecute:=FALSE;
			homeStep:=homeStep+10;
		END_IF
		IF axisError THEN
			homeStep:=1460;//Error
		END_IF
	1020:
		IF 0=axis.NcToPlc.AxisState AND NOT busy AND NOT mcBusy AND 0=stopStep THEN
			homeStep:=homeStep+10;
		END_IF
	1030:
		velVelocity:=HMIItf.goHomeVelSlow;
		velDirection:=FALSE;
		velExecute:=TRUE;
		homeStep:=homeStep+10;
	1040:
		IF (bPLimitSwitch) THEN
			velExecute:=FALSE;
			homeStep:=homeStep+10;
		END_IF
		IF axisError OR (NOT bNLimitSwitch) THEN
			homeStep:=1460;//Error
		END_IF
	1050:
		IF 0=axis.NcToPlc.AxisState AND NOT busy AND NOT mcBusy AND 0=stopStep THEN
			homeStep:=homeStep+10;
		END_IF
	1060:
		homeStep:=homeStep+10;
	1070:
		goHomeRelDistance:=-ABS(homeLimitSwitch_To_DOGDistance);
		goHomeRelVelocity:=HMIItf.goHomeVel;
		mcRel(
			Axis:=axis , 
			Execute:=FALSE , );
		goHomeDelayTon(in:=FALSE);
		homeStep:=homeStep+10;
	1080:
		mcRel(
			Axis:=axis , 
			Execute:=TRUE , 
			Distance:=goHomeRelDistance , 
			Velocity:=goHomeRelVelocity , 
			Acceleration:=relAcceleration , 
			Deceleration:=relDeceleration , 
			Jerk:= relJerk, 
			BufferMode:= , 
			Options:= , 
			Done=> , 
			Busy=> , 
			Active=> , 
			CommandAborted=> , 
			Error=> , 
			ErrorID=> );
		IF mcRel.Done THEN
			homeStep:=homeStep+10;
		END_IF
		IF axisError OR mcRel.Error OR mcRel.ErrorID<>0 THEN
			homeStep:=1460;//Error
		END_IF
	1090:
		goHomeDelayTon(IN:=NOT goHomeDelayTon.Q, PT:=T#500MS);
		IF goHomeDelayTon.Q THEN
			goHomeDelayTon(in:=FALSE);
			homeStep:=homeStep+10;
		END_IF
		mcRel(
			Axis:=axis , 
			Execute:=FALSE , );
		mcSetPos(
		      Axis:=axis , 
		      Execute:=FALSE , );
	1100:
		mcSetPos(
			Axis:=axis , 
			Execute:=TRUE , 
			Position:=0 , 
			Mode:= , 
			Options:= setPosOptions, 
			Done=> , 
			Busy=> , 
			Error=> , 
			ErrorID=> );
		IF mcSetPos.Done THEN
			homeStep:=homeStep+10;
	   	END_IF
		IF axisError OR mcSetPos.Error OR mcSetPos.ErrorID<>0 THEN
			homeStep:=1460;//Error
		END_IF
	1110:
	 	mcSetPos(
		      Axis:=axis , 
		      Execute:=FALSE , );
		homeStep:=homeStep+10;
	1120:
		homeStep:=1450;//Done
	 
	1450://Home Done
		homeStep:=0;
		homeBusy:=FALSE;
		homeDone:=TRUE;
		homeErrorDone:=FALSE;
		axisHomeState:=TRUE;
		
		homeExecute:=FALSE;
		
	1460://Home Error
		homeStep:=0;
		homeBusy:=FALSE;
		homeDone:=FALSE;
		homeErrorDone:=TRUE;
		axisHomeState:=FALSE;
		
		homeExecute:=FALSE;
		
		errorStep:=6;

(************** 负限位做原点 ********************)
	2000://负方向回原点开始，以负限位做原点
		goHomeDelayTon(in:=(0=stopStep ), PT:=T#500MS);
		IF 0=axis.NcToPlc.AxisState AND NOT busy AND NOT mcBusy AND 0=stopStep AND goHomeDelayTon.Q THEN
			goHomeDelayTon(in:=FALSE);
			homeStep:=homeStep+10;
		END_IF
	2010://负限位信号
		velVelocity:=HMIItf.goHomeVel;
		velDirection:=FALSE;
		velExecute:=TRUE;
		IF (NOT bNLimitSwitch) THEN
			velExecute:=FALSE;
			homeStep:=homeStep+10;
		END_IF
		IF axisError THEN
			homeStep:=2460;//Error
		END_IF
	2020:
		IF 0=axis.NcToPlc.AxisState AND NOT busy AND NOT mcBusy AND 0=stopStep THEN
			homeStep:=homeStep+10;
		END_IF
	2030:
		velVelocity:=HMIItf.goHomeVelSlow;
		velDirection:=TRUE;
		velExecute:=TRUE;
		homeStep:=homeStep+10;
	2040:
		IF (bNLimitSwitch) THEN
			velExecute:=FALSE;
			homeStep:=homeStep+10;
			mcReset(//陈培华
				Axis:= axis, 
				Execute:= FALSE,
				Done=> , 
				Busy=> , 
				Error=> , 
				ErrorID=> );
		END_IF
		IF axisError OR (NOT bPLimitSwitch) THEN
			homeStep:=2460;//Error
		END_IF
	2050:
		IF 0=axis.NcToPlc.AxisState AND NOT busy AND NOT mcBusy AND 0=stopStep THEN
			homeStep:=homeStep+10;
		END_IF
	2060:
		homeStep:=homeStep+10;
	2070:
		goHomeRelDistance:=ABS(homeLimitSwitch_To_DOGDistance);
		goHomeRelVelocity:=HMIItf.goHomeVel;
		mcRel(
			Axis:=axis , 
			Execute:=FALSE , );
		goHomeDelayTon(in:=FALSE);
		homeStep:=homeStep+10;
	2080:
		mcRel(
			Axis:=axis , 
			Execute:=TRUE , 
			Distance:=goHomeRelDistance , 
			Velocity:=goHomeRelVelocity , 
			Acceleration:=relAcceleration , 
			Deceleration:=relDeceleration , 
			Jerk:= relJerk, 
			BufferMode:= , 
			Options:= , 
			Done=> , 
			Busy=> , 
			Active=> , 
			CommandAborted=> , 
			Error=> , 
			ErrorID=> );
		IF mcRel.Done THEN
			homeStep:=homeStep+10;
		END_IF
		IF axisError OR mcRel.Error OR mcRel.ErrorID<>0 THEN
			homeStep:=2460;//Error
		END_IF
	2090:
		goHomeDelayTon(IN:=NOT goHomeDelayTon.Q, PT:=T#500MS);
		IF goHomeDelayTon.Q THEN
			goHomeDelayTon(in:=FALSE);
			homeStep:=homeStep+10;
		END_IF
		mcRel(
			Axis:=axis , 
			Execute:=FALSE , );
		mcSetPos(
		      Axis:=axis , 
		      Execute:=FALSE , );
	2100:
		mcSetPos(
			Axis:=axis , 
			Execute:=TRUE , 
			Position:=0 , 
			Mode:= , 
			Options:= setPosOptions, 
			Done=> , 
			Busy=> , 
			Error=> , 
			ErrorID=> );
		IF mcSetPos.Done THEN
			homeStep:=homeStep+10;
	   	END_IF
		IF axisError OR mcSetPos.Error OR mcSetPos.ErrorID<>0 THEN
			homeStep:=2460;//Error
		END_IF
	2110:
	 	mcSetPos(
		      Axis:=axis , 
		      Execute:=FALSE , );
		homeStep:=homeStep+10;
	2120:
		homeStep:=2450;//Done
	 
	2450://Home Done
		homeStep:=0;
		homeBusy:=FALSE;
		homeDone:=TRUE;
		homeErrorDone:=FALSE;
		axisHomeState:=TRUE;
		
		homeExecute:=FALSE;
		
	2460://Home Error
		homeStep:=0;
		homeBusy:=FALSE;
		homeDone:=FALSE;
		homeErrorDone:=TRUE;
		axisHomeState:=FALSE;
		
		homeExecute:=FALSE;
		
		errorStep:=6;

(************** 只有原点信号, 执行往复搜寻动作 ********************)
	3000://and 0=stopstep加入的目的是为了防止在step=0时，触发了stop=true，且stop步骤刷新需要好几个周期，而在homestep中会立马跳转到3000步，紧接着触发mcreal,即在停止的动作指令中再去动作则会报错
		//同时，marimba项目在凸轮回原时，会在低速找零DOG时，会因为设置的慢速速度过快，导致周期时间内，捕捉不到原点信号，机台会慢速朝一个方向不停运动
		IF 0=axis.NcToPlc.AxisState AND NOT busy AND NOT mcBusy AND 0=stopstep  THEN
			homeStep:=homeStep+10;
		END_IF
	3010:
		mcRel(
			Axis:=axis , 
			Execute:=FALSE , );
		homeStep:=homeStep+10;
	3020:
		IF homeDirection THEN
	       goHomeRelDistance:=1*ABS(homeOnlyDOGDistance);
        ELSE
	       goHomeRelDistance:=-1*ABS(homeOnlyDOGDistance);
        END_IF
		goHomeRelVelocity:=HMIItf.goHomeVel;
		homeStep:=3210;
	
	3100://开始搜寻
		IF ABS(goHomeRelDistance)>ABS(homeOnlyDOGMaxDistance) THEN
			homeStep:=3460;//Error
		ELSE
			homeStep:=homeStep+10;
		END_IF
		mcRel(
			Axis:=axis , 
			Execute:=FALSE , );
	3110:
		mcRel(
			Axis:=axis , 
			Execute:=TRUE , 
			Distance:=20*goHomeRelDistance , 
			Velocity:=goHomeRelVelocity , 
			Acceleration:=relAcceleration , 
			Deceleration:=relDeceleration , 
			Jerk:= relJerk, 
			BufferMode:= , 
			Options:= , 
			Done=> , 
			Busy=> , 
			Active=> , 
			CommandAborted=> , 
			Error=> , 
			ErrorID=> );
		IF mcRel.Done THEN
			homeStep:=3120;
		END_IF
		goHomeTrigF1(CLK:=(DOGPointSwitch));
		IF goHomeTrigF1.Q THEN
			stopExecute:=TRUE;
			IF goHomeRelDistance>0 THEN
				homeStep:=3200;//创造 mcHome 执行条件
			ELSE
				homeStep:=3300;//mcHome 执行
			END_IF
		END_IF
		IF axisError OR mcRel.Error OR mcRel.ErrorID<>0 THEN
			homeStep:=3460;//Error
		END_IF
	3120:
		IF goHomeRelDistance>0 THEN
			goHomeRelDistance:=1*(ABS(goHomeRelDistance)+ABS(homeOnlyDOGDistance));//
		ELSE
			goHomeRelDistance:=-1*(ABS(goHomeRelDistance)+ABS(homeOnlyDOGDistance));//
		END_IF
		goHomeRelVelocity:=HMIItf.goHomeVel;
		homeStep:=3100;//反向搜寻
	
	3200://创造 mcHome 执行条件
		IF 0=axis.NcToPlc.AxisState AND NOT busy AND NOT mcBusy AND 0=stopStep THEN
			homeStep:=homeStep+10;
		END_IF
	3210:
		velVelocity:=HMIItf.goHomeVel;
		velDirection:=NOT homeDirection;
		velExecute:=TRUE;
		homeStep:=homeStep+10;
	3220:
		goHomeTrigF1(CLK:=(DOGPointSwitch));
		IF goHomeTrigF1.Q THEN
			velExecute:=FALSE;
			homeStep:=homeStep+10;
		END_IF
		IF axisError THEN
			homeStep:=3460;//Error
		END_IF
	3230:
		homeStep:=3300;//mcHome 执行
	
	3300://mcHome 执行
		IF 0=axis.NcToPlc.AxisState AND NOT busy AND NOT mcBusy THEN
			homeStep:=homeStep+10;
		END_IF
	3310:
		homeStep:=homeStep+10;
		mcHome(
			Axis:= axis, 
			Execute:= FALSE,  
			HomingMode:= );//MC_DefaultHoming  MC_Direct
	3320:
		powerEnable_Inner:=FALSE;
		goHomeDelayTon(in:=NOT goHomeDelayTon.Q,PT:=T#800MS);
		IF goHomeDelayTon.Q AND NOT powerReady THEN
			homeStep:=homeStep+10;
			goHomeDelayTon(in:=FALSE);
		END_IF
	3330:
		homeStep:=homeStep+10;
	3340:
		powerEnable_Inner:=TRUE;
		goHomeDelayTon(in:=NOT goHomeDelayTon.Q,PT:=T#800MS);
		IF goHomeDelayTon.Q AND powerReady THEN
			homeStep:=homeStep+10;
			goHomeDelayTon(in:=FALSE);
		END_IF
	3350:
		homeStep:=homeStep+10;
	3360:
		homeStep:=homeStep+10;
	3370:
		mcHome(
			Axis:=axis , 
			Execute:=TRUE , 
			Position:=homePosition , 
			HomingMode:= , //MC_DefaultHoming  MC_Direct
			BufferMode:= , 
			Options:= , 
			bCalibrationCam:= DOGPointSwitch, 
			Done=> , 
			Busy=> , 
			Active=> , 
			CommandAborted=> , 
			Error=> , 
			ErrorID=> );
		IF (*NOT mcHome.Busy*) mcHome.Done AND NOT mcHome.Error THEN
			mcHome(
				Axis:= axis, 
				Execute:= FALSE, 
				HomingMode:= );//MC_DefaultHoming  MC_Direct
			homeStep:=homeStep+10;
		ELSIF mcHome.Error THEN
			homeStep:=3460;//Home Error
		END_IF
	3380:
		goHomeDelayTon(in:=NOT goHomeDelayTon.Q,PT:=T#500MS);
		IF goHomeDelayTon.Q THEN
			goHomeDelayTon(in:=FALSE);
			homeStep:=homeStep+10;
		END_IF
	3390:
		homeStep:=homeStep+10;
		(*mcSetPos(
			Axis:=axis , 
			Execute:=TRUE , 
			Position:=homePosition);
		goHomeDelayTon(in:=NOT goHomeDelayTon.Q,PT:=T#1000MS);//HMIItf.goHomeDelayTime
		IF goHomeDelayTon.Q THEN
			goHomeDelayTon(in:=FALSE);
			homeStep:=homeStep+10;
		END_IF*)
	3400:
		IF ABS(axis.NcToPlc.ActPos)<homeCheckRange THEN
			homeStep:=3450;//Done
		ELSE
			homeStep:=3460;//Error
		END_IF

	3450://Home Done
		homeStep:=0;
		homeBusy:=FALSE;
		homeDone:=TRUE;
		homeErrorDone:=FALSE;
		axisHomeState:=TRUE;
		
		homeExecute:=FALSE;
		
	3460://Home Error
		homeStep:=0;
		homeBusy:=FALSE;
		homeDone:=FALSE;
		homeErrorDone:=TRUE;
		axisHomeState:=FALSE;
		
		homeExecute:=FALSE;
		
		errorStep:=6;
		
(************** Error step ********************)
	50000://Error step
		stopExecute:=TRUE;
		homeStep:=homeStep+1;
	50001://reset status
		IF 0=axis.NcToPlc.AxisState AND NOT busy THEN
			homeStep:=0;
			homeBusy:=FALSE;
			homeDone:=FALSE;
			homeErrorDone:=TRUE;
			axisHomeState:=FALSE;
			
			homeExecute:=FALSE;
		END_IF
END_CASE
END_ACTION

ACTION InitHMI_ACT:
//将HMI上的数据和轴关联起来
HMIItf.actualPos:=axisActualPos;//HMI实际位置
HMIItf.actualVel:=axisActualVel;//HMI实际速率
HMIItf.forwardLimitSwitch:=bPLimitSwitch AND bSoftPLimit;
HMIItf.backwardsLimitSwitch:=bNLimitSwitch AND bSoftNLimit;
HMIItf.dogPointSwitch:=DOGPointSwitch;
HMIItf.forwardEnable:=powerEnable_Positive;
HMIItf.backwardsEnable:=powerEnable_Negative;
HMIItf.powerEnable:=powerReady;
HMIItf.running:=busy AND ABS(axisActualVel)>0.01;
HMIItf.jogNrunning:=jogBusy AND HMIItf.running AND (axisActualVel)<0;
HMIItf.jogPrunning:=jogBusy AND HMIItf.running AND (axisActualVel)>0;
HMIItf.velNrunning:=velBusy AND HMIItf.running AND (axisActualVel)<0;
HMIItf.velPrunning:=velBusy AND HMIItf.running AND (axisActualVel)>0;
HMIItf.busy:=axisBusy;
HMIItf.done:=axisDone;
HMIItf.error:=axisError;
HMIItf.oPause:=axisPause;
HMIItf.errID:=UDINT_TO_DINT(axisErrId);
HMIItf.errTxt:=axisErrTxt;
HMIItf.errWTxt:=axisErrWTxt;
HMIItf.PTPErrID:=PTPErrID;
HMIItf.enable:=axisEnable;
//HMIItf.softPLimitPos:=;
//HMIItf.softNLimitPos:=;
HMIItf.ctrlModeCondition:=hmiEN;//(ctrlMode=ControlMode.eManualCtrMode);
HMIItf.jogCondition:=jogCondition;
HMIItf.velCondition:=velCondition;
HMIItf.relCondition:=relCondition AND 0=loopStep;
HMIItf.absCondition:=absCondition AND 0=loopStep;
HMIItf.homeCondition:=homeCondition;
HMIItf.loopRelCondition:=relCondition AND 0=loopStep;
HMIItf.loopAbsCondition:=absCondition AND 0=loopStep;
HMIItf.loopHomeToAbsCondition:=absCondition AND 0=loopStepHome;
HMIItf.setCondition:=setCondition;
IF NOT bInit THEN
	HMIItf.goHomeVel:=homeVel;
	HMIItf.goHomeVelSlow:=homeVelSlow;
	HMIItf.softPLimitPos:=softPLimitPos;
	HMIItf.softNLimitPos:=softNLimitPos;
END_IF
//HMIItf.goHomeDrtInv:=homeDirection;//取消
HMIItf.goHomeDone:=axisHomeState;
HMIItf.nameTXT:=nameTXT;

noteTON_P(IN:=note_abs,PT:=T#0.1S);
noteRTrig_P(CLK:=noteTON_P.Q);
IF noteRTrig_P.Q THEN
//	gLog_Note.append_EX(noteWTXT_abs);
END_IF
noteTON_N(IN:=note_jog,PT:=T#0.1S);
noteRTrig_N(CLK:=noteTON_N.Q);
IF noteRTrig_N.Q THEN
//	gLog_Note.append_EX(noteWTXT_jog);
END_IF
END_ACTION

ACTION JogMove_ACT:
//轴JOG运行控制--jogExecute触发条件是切换型
IF NOT bE_Stop THEN
	jogStep:=0;
	jogExecute:=FALSE;
END_IF
jogCondition:=(NOT axisError AND NOT axisStopFlag 
				AND NOT axisBusy AND powerReady 
				AND jogConditionOuter AND bE_Stop AND NOT axisPause);

mcJog(
	Axis:=axis , 
	JogForward:= , 
	JogBackwards:= , 
	Mode:=MC_JOGMODE_CONTINOUS, //MC_JOGMODE_STANDARD_SLOW, MC_JOGMODE_STANDARD_FAST, MC_JOGMODE_CONTINOUS, MC_JOGMODE_INCHING, MC_JOGMODE_INCHING_MODULO
	Position:= , 
	Velocity:= , 
	Acceleration:= , 
	Deceleration:= , 
	Jerk:= , 
	Done=> , 
	Busy=> , 
	Active=> , 
	CommandAborted=> , 
	Error=> , 
	ErrorID=> );

CASE jogStep OF
0:
	jogBusy:=FALSE;
	IF jogExecute AND (NOT jogCondition OR NOT powerEnable_Negative OR NOT powerEnable_Positive  OR jogVelocity>0.2) THEN
		note_abs:=FALSE;
		note_jog:=TRUE;
		note_vel:=FALSE;
		note_home:=FALSE;
		note_rel:=FALSE;
	END_IF
	IF jogExecute AND jogCondition THEN
		note_abs:=FALSE;
		note_jog:=FALSE;
		note_vel:=FALSE;
		note_home:=FALSE;
		note_rel:=FALSE;
		jogBusy:=TRUE;
		jogDone:=FALSE;
		jogErrorDone:=FALSE;
		IF jogDirection THEN
			jogForward:=TRUE;
			jogBackwards:=FALSE;
		ELSE
			jogForward:=FALSE;
			jogBackwards:=TRUE;
		END_IF
		jogStep:=10;
		mcReset(
				Axis:= axis, 
				Execute:= TRUE,
				Done=> , 
				Busy=> , 
				Error=> , 
				ErrorID=> );
	ELSE
		jogExecute:=FALSE;
	END_IF
	mcJog(
		Axis:=axis , 
		JogForward:=FALSE , 
		JogBackwards:=FALSE ,);
10:
	IF NOT axisStopFlag AND powerReady AND 0=stopStep THEN
		jogStep:=20;
		mcReset(//陈培华
				Axis:= axis, 
				Execute:= FALSE,
				Done=> , 
				Busy=> , 
				Error=> , 
				ErrorID=> );
	END_IF
20:
	IF jogDirection THEN
		IF NOT bPLimitSwitch OR NOT bSoftPLimit OR NOT powerEnable_Positive THEN
			axisStopFlag:=TRUE;

			IF NOT bPLimitSwitch THEN
				errorStep:=3;
			END_IF
			IF NOT bSoftPLimit THEN
				errorStep:=2;
			END_IF
			IF NOT powerEnable_Positive THEN
				errorStep:=19;
			END_IF
			jogStep:=10000;//error
			RETURN;
		END_IF
	ELSE
		IF NOT bNLimitSwitch OR NOT bSoftNLimit OR NOT powerEnable_Negative THEN
			axisStopFlag:=TRUE;

			IF NOT bNLimitSwitch THEN
				errorStep:=4;
			END_IF
			IF NOT bSoftNLimit THEN
				errorStep:=2;
			END_IF
			IF NOT powerEnable_Negative THEN
				errorStep:=19;
			END_IF
			jogStep:=10000;//error
			RETURN;
		END_IF
	END_IF
	
	mcJog(
		Axis:=axis , 
		JogForward:=jogForward , 
		JogBackwards:=jogBackwards , 
		Mode:=MC_JOGMODE_CONTINOUS, //MC_JOGMODE_STANDARD_SLOW, MC_JOGMODE_STANDARD_FAST, MC_JOGMODE_CONTINOUS, MC_JOGMODE_INCHING, MC_JOGMODE_INCHING_MODULO
		Position:= , 
		Velocity:=jogVelocity , 
		Acceleration:=jogAcceleration , 
		Deceleration:=jogDeceleration , 
		Jerk:=jogJerk , 
		Done=> , 
		Busy=> , 
		Active=> , 
		CommandAborted=> , 
		Error=> , 
		ErrorID=> );
	IF NOT jogExecute THEN
		jogStep:=5000;//done
	END_IF
	IF mcJog.Error OR mcJog.ErrorID<>0 THEN
		errorStep:=8;
		jogStep:=10000;//error
	END_IF

	IF axisStopFlag OR NOT powerReady OR 0<>stopStep THEN
		jogStep:=4000;//stop
	END_IF

4000://Stop
	mcJog(
		Axis:=axis , 
		JogForward:=FALSE , 
		JogBackwards:=FALSE ,);
	jogExecute:=FALSE;
	jogBusy:=FALSE;
	jogDone:=FALSE;
	jogErrorDone:=FALSE;
	jogStep:=0;
5000://Done
	mcJog(
		Axis:=axis , 
		JogForward:=FALSE , 
		JogBackwards:=FALSE ,);
	jogExecute:=FALSE;
	jogBusy:=FALSE;
	jogDone:=TRUE;
	jogErrorDone:=FALSE;
	jogStep:=0;
10000://Error
	mcJog(
		Axis:=axis , 
		JogForward:=FALSE , 
		JogBackwards:=FALSE ,);
	jogExecute:=FALSE;
	jogBusy:=FALSE;
	jogDone:=FALSE;
	jogErrorDone:=TRUE;
	jogStep:=0;
END_CASE
END_ACTION

ACTION LoopHomeToPos_ACT:
IF loopGoHome AND loopStepHome=0 THEN
	loopCycleTimes:=0;
	loopFirstPoint:=HMIItf.loopFirstPoint;
	loopGoVel:=HMIItf.loopGoVel;
	loopCycle:=HMIItf.loopCycle;
	loopStepHome:=1000;//相对运动 Loop
END_IF
IF NOT bE_Stop OR axisStopFlag THEN
	loopStepHome:=0;
	tHomeTemp(IN:=FALSE);
	loopWatingTON(IN:=FALSE);
END_IF
loopGoHome:=FALSE;
CASE loopStepHome OF
0:
	//Ready


//相对运动 Loop
1000:
	IF homeCondition THEN
		loopStepHome:=loopStepHome+10;
		tHomeTemp(IN:=FALSE);
	END_IF
1010:
	homeExecute:=TRUE;
	loopStepHome:=loopStepHome+10;
1020:
	tHomeTemp(IN:=NOT tHomeTemp.Q, PT:=T#50MS);
	IF tHomeTemp.Q THEN
		tHomeTemp(IN:=FALSE);
		loopStepHome:=loopStepHome+10;
	END_IF
	
1030:
	IF homeDone THEN
		loopStepHome:=loopStepHome+10;
	END_IF
1040:
	IF absCondition THEN
		loopStepHome:=loopStepHome+10;
	END_IF
1050:
	absVelocity:=loopGoVel;
	absPosition:=loopFirstPoint;
	absExecute:=TRUE;
	IF absBusy THEN
		absExecute:=FALSE;
		loopStepHome:=loopStepHome+10;
	END_IF
1060:
	IF NOT absBusy AND absDone THEN
		loopStepHome:=loopStepHome+10;
		loopCycleTimes:=loopCycleTimes+1;
	END_IF
	IF axisError THEN
		loopStepHome:=10000;//Error
	END_IF
	tHomeTemp(IN:=FALSE);
1070:
	loopWatingTON(IN:=NOT loopWatingTON.Q, PT:=UINT_TO_TIME(HMIItf.loopWatingTime));
	IF loopWatingTON.Q THEN
		loopWatingTON(IN:=FALSE);
		loopStepHome:=loopStepHome+10;
	END_IF
1080:
	IF (0=loopCycleTimes) OR loopCycle<=loopCycleTimes THEN
		loopStepHome:=8000;//Done
	ELSE
		loopStepHome:=1000;
	END_IF



//Done
8000:
	loopStepHome:=0;

//Error
10000:
	loopStepHome:=0;
END_CASE
END_ACTION

ACTION LoopMove_ACT:
IF loopRelGo AND relCondition AND 0=loopStep THEN
	loopFirstPoint:=HMIItf.loopFirstPoint;
	loopSecondPoint:=HMIItf.loopSecondPoint;
	loopGoVel:=HMIItf.loopGoVel;
	loopCycle:=HMIItf.loopCycle;
	loopWatingTime:=HMIItf.loopWatingTime;
	
	loopCycleTimes:=0;
	loopStep:=1000;//相对运动 Loop
END_IF
IF loopAbsGo AND absCondition AND 0=loopStep THEN
	loopFirstPoint:=HMIItf.loopFirstPoint;
	loopSecondPoint:=HMIItf.loopSecondPoint;
	loopGoVel:=HMIItf.loopGoVel;
	loopCycle:=HMIItf.loopCycle;
	loopWatingTime:=HMIItf.loopWatingTime;
	
	loopCycleTimes:=0;
	loopStep:=3000;//绝对运动 Loop
END_IF
loopRelGo:=FALSE;
loopAbsGo:=FALSE;

IF NOT bE_Stop OR axisStopFlag THEN
	loopStep:=0;
END_IF

CASE loopStep OF
0:
	//Ready


//相对运动 Loop
1000:
	IF relCondition THEN
		loopStep:=loopStep+10;
	END_IF
1010:
	IF (0=loopCycle) OR loopCycle<=loopCycleTimes THEN
		loopStep:=8000;//Done
	ELSE
		loopCycleTimes:=loopCycleTimes+1;
		loopStep:=loopStep+10;
	END_IF
1020:
	relVelocity:=loopGoVel;
	relDistance:=loopFirstPoint;
	relExecute:=TRUE;
	IF relBusy THEN
		relExecute:=FALSE;
		loopStep:=loopStep+10;
	END_IF
1030:
	IF NOT relBusy AND relDone THEN
		loopStep:=loopStep+10;
	END_IF
	IF axisError THEN
		loopStep:=10000;//Error
	END_IF
	loopWatingTON(IN:=FALSE);
1040:
	loopWatingTON(IN:=NOT loopWatingTON.Q, PT:=UINT_TO_TIME(loopWatingTime));
	IF loopWatingTON.Q AND relCondition THEN
		loopWatingTON(IN:=FALSE);
		loopStep:=loopStep+10;
	END_IF
1050:
	relVelocity:=loopGoVel;
	relDistance:=loopSecondPoint;
	relExecute:=TRUE;
	IF relBusy THEN
		relExecute:=FALSE;
		loopStep:=loopStep+10;
	END_IF
1060:
	IF NOT relBusy AND relDone THEN
		loopStep:=loopStep+10;
	END_IF
	IF axisError THEN
		loopStep:=10000;//Error
	END_IF
	loopWatingTON(IN:=FALSE);
1070:
	loopWatingTON(IN:=NOT loopWatingTON.Q, PT:=UINT_TO_TIME(loopWatingTime));
	IF loopWatingTON.Q THEN
		loopWatingTON(IN:=FALSE);
		loopStep:=loopStep+10;
	END_IF
1080:
	IF (0=loopCycle) OR loopCycle<=loopCycleTimes THEN
		loopStep:=8000;//Done
	ELSE
		loopStep:=1000;
	END_IF


//绝对运动 Loop
3000:
	IF absCondition THEN
		loopStep:=loopStep+10;
	END_IF
3010:
	IF (0=loopCycle) OR loopCycle<=loopCycleTimes THEN
		loopStep:=8000;//Done
	ELSE
		loopCycleTimes:=loopCycleTimes+1;
		loopStep:=loopStep+10;
	END_IF
3020:
	absVelocity:=loopGoVel;
	absPosition:=loopFirstPoint;
	absExecute:=TRUE;
	IF absBusy THEN
		absExecute:=FALSE;
		loopStep:=loopStep+10;
	END_IF
3030:
	IF NOT absBusy AND absDone THEN
		loopStep:=loopStep+10;
	END_IF
	IF axisError THEN
		loopStep:=10000;//Error
	END_IF
	loopWatingTON(IN:=FALSE);
3040:
	loopWatingTON(IN:=NOT loopWatingTON.Q, PT:=UINT_TO_TIME(loopWatingTime));
	IF loopWatingTON.Q AND absCondition THEN
		loopWatingTON(IN:=FALSE);
		loopStep:=loopStep+10;
	END_IF
3050:
	absVelocity:=loopGoVel;
	absPosition:=loopSecondPoint;
	absExecute:=TRUE;
	IF absBusy THEN
		absExecute:=FALSE;
		loopStep:=loopStep+10;
	END_IF
3060:
	IF NOT absBusy AND absDone THEN
		loopStep:=loopStep+10;
	END_IF
	IF axisError THEN
		loopStep:=10000;//Error
	END_IF
	loopWatingTON(IN:=FALSE);
3070:
	loopWatingTON(IN:=NOT loopWatingTON.Q, PT:=UINT_TO_TIME(loopWatingTime));
	IF loopWatingTON.Q AND absCondition THEN
		loopWatingTON(IN:=FALSE);
		loopStep:=loopStep+10;
	END_IF
3080:
	IF (0=loopCycle) OR loopCycle<=loopCycleTimes THEN
		loopStep:=8000;//Done
	ELSE
		loopStep:=3000;
	END_IF

//Done
8000:
	loopStep:=0;

//Error
10000:
	loopStep:=0;
END_CASE
END_ACTION

ACTION ManualCtr_ACT:

//*********** Stop button ***************
stopTrigR1(CLK:=HMIItf.stop OR stoptemp);
IF stopTrigR1.Q THEN
	axisStopFlag:=TRUE;
END_IF
CASE manualStep OF
0:
	IF axisStopFlag THEN
		stopExecute:=TRUE;
		manualStep:=manualStep+1;
	END_IF
1:
	manualStep:=manualStep+1;
2:
	IF NOT axisStopFlag THEN
		manualStep:=0;
	END_IF
END_CASE
//Velo Limit
IF HMIItf.manSoftLimitVel<0 THEN
	HMIItf.manSoftLimitVel:=ABS(HMIItf.manSoftLimitVel);
END_IF
//Jog
IF HMIItf.manJogVel>HMIItf.manSoftLimitVel THEN
	HMIItf.manJogVel:=HMIItf.manSoftLimitVel;
END_IF
//manVel
IF HMIItf.manVel>HMIItf.manSoftLimitVel THEN
	HMIItf.manVel:=HMIItf.manSoftLimitVel;
END_IF
//in each mode, stop is still working
stopTon(in:=axisStopFlag,pt:=T#1S);
IF stopTon.Q THEN
	axisStopFlag:=FALSE;
	stopTon(in:=FALSE);
	stoptemp:=FALSE;
END_IF

IF (NOT axisEnable) 
	AND (HMIItf.manJogGo OR HMIItf.manRelGo OR HMIItf.manVelGo OR HMIItf.manABSGo OR HMIItf.reset OR HMIItf.stop 
		OR HMIItf.pauseB OR HMIItf.power OR HMIItf.setZero OR HMIItf.goHomeGo) THEN
	RETURN;
END_IF

//*********** Reset button ***************
resetTrigR1(CLK:=HMIItf.reset);
IF resetTrigR1.Q THEN
	resetExecute:=TRUE;
	stoptemp:=FALSE;
END_IF
//resetTrigR2(CLK:=HMIItf.reset2);
//IF resetTrigR2.Q THEN
//	resetExecute2:=TRUE;
//	stoptemp:=FALSE;
//END_IF

IF HMIItf.ctrlModeCondition THEN
//*********** Home button ***************
	goHomeTrigR1(CLK:=HMIItf.goHomeGo);
	IF goHomeTrigR1.Q AND NOT axisBusy THEN
		homeExecute:=TRUE;
	END_IF

//*********** JOG button ***************
	IF HMIItf.manJogVel<0 THEN
		HMIItf.manJogVel:=ABS(HMIItf.manJogVel);
	END_IF
	jogTrigR1_NAiko(CLK:=HMIItf.manJogN);
	jogTrigF1_NAiko(CLK:=HMIItf.manJogN);
	IF jogTrigR1_NAiko.Q THEN
		HMIItf.choiceOfDirection:=FALSE;
		jogDirection:=FALSE;
		HMIItf.manJogGo:=TRUE;
	END_IF
	IF jogTrigF1_NAiko.Q THEN
		HMIItf.manJogGo:=FALSE;
	END_IF
	jogTrigR1_PAiko(CLK:=HMIItf.manJogP);
	jogTrigF1_PAiko(CLK:=HMIItf.manJogP);
	IF jogTrigR1_PAiko.Q THEN
		HMIItf.choiceOfDirection:=TRUE;
		jogDirection:=TRUE;
		HMIItf.manJogGo:=TRUE;
	END_IF
	IF jogTrigF1_PAiko.Q THEN
		HMIItf.manJogGo:=FALSE;
	END_IF
	jogTrigR1(CLK:=HMIItf.manJogGo);
	jogTrigF1(CLK:=HMIItf.manJogGo);
	IF jogTrigR1.Q AND NOT axisBusy THEN
		IF HMIItf.choiceOfDirection THEN
			jogDirection:=TRUE;
		ELSE
			jogDirection:=FALSE;
		END_IF
		jogVelocity:=ABS(HMIItf.manJogVel);
		jogExecute:=TRUE;
	END_IF
	IF jogTrigF1.Q THEN
		jogExecute:=FALSE;
	END_IF
	
//*********** VelGo button ***************
//	velTrigR1_NAiko(CLK:=HMIItf.manVelN);
//	velTrigF1_NAiko(CLK:=HMIItf.manVelN);
//	IF velTrigR1_NAiko.Q AND NOT velBusy THEN
//		HMIItf.choiceOfDirection:=FALSE;
//		jogDirection:=FALSE;
//		HMIItf.manVelGo:=TRUE;
//	END_IF
//	IF velTrigR1_NAiko.Q AND velBusy THEN
//		HMIItf.manVelGo:=FALSE;
//		axisStopFlag:=TRUE;
//	END_IF
//	IF velTrigF1_NAiko.Q THEN
//		HMIItf.manVelGo:=FALSE;
//	END_IF
	
//	velTrigR1_PAiko(CLK:=HMIItf.manVelP);
//	velTrigF1_PAiko(CLK:=HMIItf.manVelP);
//	IF velTrigR1_PAiko.Q AND NOT velBusy THEN
//		HMIItf.choiceOfDirection:=TRUE;
//		jogDirection:=TRUE;
//		HMIItf.manVelGo:=TRUE;
//	END_IF
//	IF velTrigR1_PAiko.Q AND velBusy THEN
//		axisStopFlag:=TRUE;
//		HMIItf.manVelGo:=FALSE;
//	END_IF
//	IF velTrigF1_PAiko.Q THEN
//		HMIItf.manVelGo:=FALSE;
//	END_IF
	
	velTrigR1(CLK:=HMIItf.manVelGo);
	IF velTrigR1.Q THEN
		IF HMIItf.choiceOfDirection THEN
			velDirection:=TRUE;
		ELSE
			velDirection:=FALSE;
		END_IF
		IF velExecute THEN
			velExecute:=FALSE;
		ELSIF NOT axisBusy THEN
			velExecute:=TRUE;
		END_IF
		velVelocity:=ABS(HMIItf.manJogVel);
	END_IF
	
//*********** RelGo button ***************
	IF HMIItf.manVel<0 THEN
		HMIItf.manVel:=ABS(HMIItf.manVel);
	END_IF
	IF HMIItf.manRelDis<0 THEN
		HMIItf.manRelDis:=ABS(HMIItf.manRelDis);
	END_IF
	relT1(IN:=HMIItf.manRelGo,PT:=T#1S);
	relTrigR1(CLK:=relT1.Q);
	IF relTrigR1.Q AND NOT axisBusy THEN
		relVelocity:=ABS(HMIItf.manVel);
		IF HMIItf.choiceOfDirection THEN
			relDistance:=HMIItf.manRelDis;
		ELSE
			relDistance:=0-HMIItf.manRelDis;
		END_IF
		relExecute:=TRUE;
	END_IF

//*********** AbsGo button ***************
	absT1(IN:=HMIItf.manABSGo,PT:=T#1S);
	absTrigR1(CLK:=absT1.Q);
	IF absTrigR1.Q AND NOT axisBusy THEN
		absVelocity:=ABS(HMIItf.manVel);
		absPosition:=HMIItf.manABSPos;
		absExecute:=TRUE;
	END_IF
	absRP(CLK:=HMIItf.GoToOpen);
	IF absRP.Q AND bP_Pos<>0.777 THEN
		absVelocity:=ABS(HMIItf.manVel);
		absPosition:=bP_Pos;
		absExecute:=TRUE;
	END_IF
	absRN(CLK:=HMIItf.GoToClose);
	IF absRN.Q AND bN_Pos<>0.777 THEN
		absVelocity:=ABS(HMIItf.manVel);
		absPosition:=bN_Pos;
		absExecute:=TRUE;
	END_IF
//*********** Zero button ***************
	setPosTrigR1(CLK:=HMIItf.setZero);
	IF setPosTrigR1.Q AND NOT axisBusy THEN
		setPosPosition:=0;
		setPosExecute:=TRUE;
	END_IF
	
//*********** Power button ***************
	powerTrigF1(CLK:=HMIItf.power);
	IF powerTrigF1.Q AND NOT axisBusy THEN
		IF powerEnable THEN
			powerEnable:=FALSE;
		ELSE
			powerEnable:=TRUE;
		END_IF
	END_IF

//*********** Pause button ***************
	pause_Manual_F_Trig(CLK:=HMIItf.pauseB);
	IF pause_Manual_F_Trig.Q THEN
		pauseExecute:=NOT pauseExecute;
	END_IF
	
//*********** LOOP ***************
//*********** loopRelGo button ***************
	loopRelGoT1(IN:=HMIItf.loopRelGo,PT:=T#2S);
	loopRelGoTrigR1(CLK:=loopRelGoT1.Q);
	IF loopRelGoTrigR1.Q AND NOT axisBusy THEN
		loopRelGo:=TRUE;
	END_IF
//*********** loopAbsGo button ***************
	loopAbsGoT1(IN:=HMIItf.loopAbsGo,PT:=T#2S);
	loopAbsGoTrigR1(CLK:=loopAbsGoT1.Q);
	IF loopAbsGoTrigR1.Q AND NOT axisBusy THEN
		loopAbsGo:=TRUE;
	END_IF
	loopHomeToPosGoT1(IN:=HMIItf.loopHomeToPosGo,PT:=T#2S);
	loopHomeToPosTrigR1(CLK:=loopHomeToPosGoT1.Q);
	IF loopHomeToPosTrigR1.Q AND NOT axisBusy THEN
		loopGoHome:=TRUE;
	END_IF
ELSE
	HMIItf.manABSPos:=0;
	HMIItf.manRelDis:=0;
	
	HMIItf.manJogGo:=FALSE;
	HMIItf.manVelGo:=FALSE;
	HMIItf.manRelGo:=FALSE;
	HMIItf.manABSGo:=FALSE;
	HMIItf.pauseB:=FALSE;
	//HMIItf.power:=FALSE;//解决控制模式切换导致掉使能的问题
	HMIItf.setZero:=FALSE;
	HMIItf.goHomeGo:=FALSE;
	HMIItf.loopRelGo:=FALSE;
	HMIItf.loopAbsGo:=FALSE;
	
	relT1(IN:=FALSE);
	absT1(IN:=FALSE);
	loopRelGoT1(IN:=FALSE);
	loopAbsGoT1(IN:=FALSE);
END_IF
END_ACTION

ACTION MoveModulo_ACT:
//轴 模运动运行控制-- moveModuloExecute 触发条件是复归型
IF NOT bE_Stop THEN
	moveModuloStep:=0;
	moveModuloExecute:=FALSE;
END_IF
moveModuloCondition:=(NOT axisError AND NOT axisStopFlag 
				AND (NOT axisBusy OR 0<>loopStep) AND powerReady 
				AND moveModuloConditionOuter AND bE_Stop AND NOT axisPause);
mcMoveModulo(
	Axis:= axis, 
	Execute:= , 
	Position:= , 
	Velocity:= , 
	Acceleration:= , 
	Deceleration:= , 
	Jerk:= , 
	Direction:= , 
	BufferMode:= , 
	Options:= , 
	Done=> , 
	Busy=> , 
	Active=> , 
	CommandAborted=> , 
	Error=> , 
	ErrorID=> );

CASE moveModuloStep OF
0:
	moveModuloBusy:=FALSE;
	IF moveModuloExecute AND moveModuloCondition THEN
		moveModuloBusy:=TRUE;
		moveModuloDone:=FALSE;
		moveModuloErrorDone:=FALSE;
		moveModuloStep:=20;
	END_IF
	moveModuloExecute:=FALSE;
	mcMoveModulo(
		Axis:=axis , 
		Execute:=FALSE ,);
20:
	IF NOT bPLimitSwitch OR NOT bNLimitSwitch OR NOT bSoftPLimit OR NOT bSoftNLimit OR NOT powerEnable_Positive OR NOT powerEnable_Negative THEN
		axisStopFlag:=TRUE;

		IF NOT bPLimitSwitch THEN
			errorStep:=3;
		ELSIF NOT bNLimitSwitch THEN
			errorStep:=4;
		END_IF
		IF NOT bSoftPLimit OR NOT bSoftNLimit THEN
			errorStep:=2;
		END_IF
		IF NOT powerEnable_Positive OR NOT powerEnable_Negative THEN
			errorStep:=19;
		END_IF
		absStep:=10000;//error
		RETURN;
	END_IF
	mcMoveModulo(
		Axis:= axis, 
		Execute:= TRUE, 
		Position:= moveModuloPosition, 
		Velocity:= moveModuloVelocity, 
		Acceleration:= moveModuloAcceleration, 
		Deceleration:= moveModuloDeceleration, 
		Jerk:= moveModuloJerk, 
		Direction:= moveModuloDirection, 
		BufferMode:= , 
		Options:= , 
		Done=> , 
		Busy=> , 
		Active=> , 
		CommandAborted=> , 
		Error=> , 
		ErrorID=> );
	IF mcMoveModulo.Done THEN//mcMoveModulo.Done信号只保持一个扫描周期
		moveModuloStep:=5000;//done
	ELSIF mcMoveModulo.Error OR mcMoveModulo.ErrorID<>0 THEN
		errorStep:=9;
		moveModuloStep:=10000;//error
	END_IF

	IF axisStopFlag OR NOT powerReady OR 0<>stopStep THEN
		moveModuloStep:=4000;//stop
	END_IF
	
4000://Stop
	mcMoveModulo(
		Axis:=axis , 
		Execute:=FALSE ,);
	moveModuloExecute:=FALSE;
	moveModuloBusy:=FALSE;
	moveModuloDone:=FALSE;
	moveModuloErrorDone:=FALSE;
	moveModuloStep:=0;
5000://Done
	mcMoveModulo(
		Axis:=axis , 
		Execute:=FALSE ,);
	moveModuloExecute:=FALSE;
	moveModuloBusy:=FALSE;
	moveModuloDone:=TRUE;
	moveModuloErrorDone:=FALSE;
	moveModuloStep:=0;
10000://Error
	mcMoveModulo(
		Axis:=axis , 
		Execute:=FALSE ,);
	moveModuloExecute:=FALSE;
	moveModuloBusy:=FALSE;
	moveModuloDone:=FALSE;
	moveModuloErrorDone:=TRUE;
	moveModuloStep:=0;
END_CASE
END_ACTION

ACTION Power_ACT:
IF powerEnable_Inner AND powerEnable AND bE_Stop THEN
	mcPower(
		Axis:= axis, 
		Enable:= TRUE, 
		Enable_Positive:= powerEnable_Positive, 
		Enable_Negative:= powerEnable_Negative, 
		Override:= overrideSet, 
		BufferMode:= , 
		Options:= , 
		Status=> , 
		Busy=> , 
		Active=> , 
		Error=> , 
		ErrorID=> );
ELSE
	mcPower(
		Axis:= axis, 
		Enable:= FALSE, 
		Enable_Positive:= powerEnable_Positive, 
		Enable_Negative:= powerEnable_Negative, 
		Override:= overrideSet, 
		BufferMode:= , 
		Options:= , 
		Status=> , 
		Busy=> , 
		Active=> , 
		Error=> , 
		ErrorID=> );
END_IF
IF mcPower.Error THEN
	errorStep:=14;
END_IF
END_ACTION

ACTION RelMove_ACT:
//轴相对运动运行控制--relExecute触发条件是复归型
IF NOT bE_Stop THEN
	relStep:=0;
	relExecute:=FALSE;
END_IF
relCondition:=(NOT axisError AND NOT axisStopFlag 
				AND (NOT axisBusy OR 0<>loopStep) AND powerReady 
				AND relConditionOuter AND bE_Stop AND NOT axisPause);

mcRel(
	Axis:=axis , 
	Execute:= , 
	Distance:= , 
	Velocity:= , 
	Acceleration:= , 
	Deceleration:= , 
	Jerk:= , 
	BufferMode:= , 
	Options:= , 
	Done=> , 
	Busy=> , 
	Active=> , 
	CommandAborted=> , 
	Error=> , 
	ErrorID=> );

CASE relStep OF
0:
	relBusy:=FALSE;
	IF relExecute AND (NOT relCondition OR NOT powerEnable_Negative OR NOT powerEnable_Positive) THEN
		note_abs:=FALSE;
		note_jog:=FALSE;
		note_vel:=FALSE;
		note_home:=FALSE;
		note_rel:=TRUE;
	END_IF
	IF relExecute AND relCondition THEN
		note_abs:=FALSE;
		note_jog:=FALSE;
		note_vel:=FALSE;
		note_home:=FALSE;
		note_rel:=FALSE;
		relBusy:=TRUE;
		relDone:=FALSE;
		relErrorDone:=FALSE;
		relStep:=10;
		mcReset(
			Axis:= axis, 
			Execute:= TRUE,
			Done=> , 
			Busy=> , 
			Error=> , 
			ErrorID=> );
	END_IF
	relExecute:=FALSE;
	mcRel(
		Axis:=axis , 
		Execute:=FALSE ,);
10:
	IF NOT axisStopFlag AND powerReady AND 0=stopStep THEN
		relStep:=20;
		mcReset(//陈培华
				Axis:= axis, 
				Execute:= FALSE,
				Done=> , 
				Busy=> , 
				Error=> , 
				ErrorID=> );
	END_IF
20:
	IF NOT bPLimitSwitch OR NOT bNLimitSwitch OR NOT bSoftPLimit OR NOT bSoftNLimit OR NOT powerEnable_Positive OR NOT powerEnable_Negative THEN
		axisStopFlag:=TRUE;

		IF NOT bPLimitSwitch THEN
			errorStep:=3;
		ELSIF NOT bNLimitSwitch THEN
			errorStep:=4;
		END_IF
		IF NOT bSoftPLimit OR NOT bSoftNLimit THEN
			errorStep:=2;
		END_IF
		IF NOT powerEnable_Positive OR NOT powerEnable_Negative THEN
			errorStep:=19;
		END_IF
		absStep:=10000;//error
		RETURN;
	END_IF
	mcRel(
		Axis:=axis , 
		Execute:=TRUE , 
		Distance:=relDistance , 
		Velocity:=relVelocity , 
		Acceleration:=relAcceleration , 
		Deceleration:=relDeceleration , 
		Jerk:=relJerk , 
		BufferMode:= , 
		Options:= , 
		Done=> , 
		Busy=> , 
		Active=> , 
		CommandAborted=> , 
		Error=> , 
		ErrorID=> );
	IF mcRel.Done THEN//mcRel.Done信号只保持一个扫描周期
		relStep:=5000;//done
	ELSIF mcRel.Error OR mcRel.ErrorID<>0 THEN
		errorStep:=10;
		relStep:=10000;//error
	END_IF

	IF axisStopFlag OR NOT powerReady OR 0<>stopStep THEN
		relStep:=4000;//stop
	END_IF
	
4000://Stop
	mcRel(
		Axis:=axis , 
		Execute:=FALSE ,);
	relExecute:=FALSE;
	relBusy:=FALSE;
	relDone:=FALSE;
	relErrorDone:=FALSE;
	relStep:=0;
5000://Done
	mcRel(
		Axis:=axis , 
		Execute:=FALSE ,);
	relExecute:=FALSE;
	relBusy:=FALSE;
	relDone:=TRUE;
	relErrorDone:=FALSE;
	relStep:=0;
10000://Error
	mcRel(
		Axis:=axis , 
		Execute:=FALSE ,);
	relExecute:=FALSE;
	relBusy:=FALSE;
	relDone:=FALSE;
	relErrorDone:=TRUE;
	relStep:=0;
END_CASE
END_ACTION

ACTION Reset_ACT:
(*
CASE resetStep OF
	0:
	IF resetExecute THEN
		resetExecute:=FALSE;
		mcReset(
			Axis:= axis, 
			Execute:= FALSE,
			Done=> , 
			Busy=> , 
			Error=> , 
			ErrorID=> );
		resetStep:=1;
	END_IF
	1:
	IF (mcError OR axis.Status.Error OR 0<>axis.NcToPlc.ErrorCode OR homeBusy) THEN
		mcReset(
			Axis:= axis, 
			Execute:= TRUE,
			Done=> , 
			Busy=> , 
			Error=> , 
			ErrorID=> );
	END_IF
	resetExecute:=FALSE;
	motorError:=FALSE;
	resetStep:=0;
END_CASE
*)
mcReset(
	Axis:= axis, 
	Execute:= ,
	Done=> , 
	Busy=> , 
	Error=> , 
	ErrorID=> );
	IF resetExecute  THEN
		note_abs:=FALSE;
		note_jog:=FALSE;
		note_vel:=TRUE;
		note_home:=FALSE;
		note_rel:=FALSE;
		mcReset(
			Axis:= axis, 
			Execute:= FALSE,
			Done=> , 
			Busy=> , 
			Error=> , 
			ErrorID=> );
		IF (mcError OR axis.Status.Error 
			OR 0<>axis.NcToPlc.ErrorCode 
			OR (homeBusy AND MotorType_DDmotor_HC=motorType)) THEN
			mcReset(
				Axis:= axis, 
				Execute:= TRUE,
				Done=> , 
				Busy=> , 
				Error=> , 
				ErrorID=> );
				//陈培华 0903
//				mcReset(
//					Axis:= axis, 
//					Execute:= FALSE,
//					Done=> , 
//					Busy=> , 
//					Error=> , 
//					ErrorID=> );
		END_IF
		motorError:=FALSE;
		errorStep:=0;
		resetExecute:=FALSE;
	ELSE
		IF resetStep=0 THEN
			mcReset(
				Axis:= axis, 
				Execute:=FALSE ,
				Done=> , 
				Busy=> , 
				Error=> , 
				ErrorID=> );
		END_IF
	END_IF
	IF mcReset.Error THEN
		errorStep:=15;
	END_IF
END_ACTION

ACTION ResetEx_ACT:
mcReset(
	Axis:= axis, 
	Execute:= ,
	Done=> , 
	Busy=> , 
	Error=> , 
	ErrorID=> );
CASE resetStep OF
	0:
		resetBusy:=FALSE;
		IF resetExecute2 THEN
			resetBusy:=TRUE;
			resetDone:=FALSE;
			resetErrorDone:=FALSE;
			resetStep:=10;
			mcReset(
				Axis:= axis, 
				Execute:= FALSE,
				Done=> , 
				Busy=> , 
				Error=> , 
				ErrorID=> );
		END_IF
		resetExecute2:=FALSE;
	10:
		mcReset(
			Axis:= axis, 
			Execute:= TRUE,
			Done=> , 
			Busy=> , 
			Error=> , 
			ErrorID=> );
		IF NOT mcReset.Busy THEN
			resetStep:=20;
			mcReset(
				Axis:= axis, 
				Execute:= FALSE,
				Done=> , 
				Busy=> , 
				Error=> , 
				ErrorID=> );
		END_IF
	20:
		resetStep:=resetStep+10;
	30:
		resetExecute:=TRUE;
		resetStep:=resetStep+10;
	40:
		resetStep:=resetStep+10;
	50:
		resetStep:=resetStep+10;
	60:
		resetBusy:=FALSE;
		resetDone:=TRUE;
		resetErrorDone:=FALSE;
		resetStep:=0;
END_CASE
END_ACTION

//设定绝对定位运行模式的位置和速度
METHOD setAbs
VAR_INPUT
	pos:LREAL;//绝对目标设定
	vel:LREAL;//速度设定
END_VAR
absPosition:=pos;
absVelocity:=vel;
END_METHOD

ACTION SetPause_ACT:
IF axisOverride<>overrideSet AND ((overrideSet<>0) OR NOT pauseExecute) THEN
	overrideSet:=axisOverride;
END_IF

pauseR_Trig(CLK:=pauseExecute);
IF pauseR_Trig.Q THEN
	overrideTemp:=overrideSet;
	overrideSet:=0;
	axisPause:=TRUE;
END_IF

pauseF_Trig(CLK:=pauseExecute);
IF pauseF_Trig.Q THEN
	overrideSet:=overrideTemp;
	axisPause:=FALSE;
	HMIItf.pauseB:=FALSE;
END_IF
END_ACTION

ACTION SetPosition_ACT:
//轴当前位置修改--setPosExecute触发条件是复归型
IF NOT bE_Stop THEN
	setPosStep:=0;
	setPosExecute:=FALSE;
END_IF
setCondition:=(NOT axisError AND NOT axisStopFlag 
				AND NOT axisBusy AND powerReady 
				AND setConditionOuter AND bE_Stop AND NOT axisPause);

mcSetPos(
	Axis:=axis , 
	Execute:= , 
	Position:= , 
	Mode:= , 
	Options:= , 
	Done=> , 
	Busy=> , 
	Error=> , 
	ErrorID=> );

CASE setPosStep OF
0:
	setPosBusy:=FALSE;
	IF setPosExecute AND (setCondition OR homeBusy) THEN
		setPosBusy:=TRUE;
		setPosDone:=FALSE;
		setPosErrorDone:=FALSE;
		
		setPosStep:=20;
	END_IF
	setPosExecute:=FALSE;
	mcSetPos(
		Axis:=axis , 
		Execute:=FALSE ,);
20:
	IF NOT bPLimitSwitch OR NOT bNLimitSwitch OR NOT bSoftPLimit OR NOT bSoftNLimit THEN
		axisStopFlag:=TRUE;

		IF NOT bPLimitSwitch THEN
			errorStep:=3;
		ELSIF NOT bNLimitSwitch THEN
			errorStep:=4;
		END_IF
		IF NOT bSoftPLimit OR NOT bSoftNLimit THEN
			errorStep:=2;
		END_IF
		
		setPosStep:=10000;//error
		RETURN;
	END_IF
	mcSetPos(
		Axis:=axis , 
		Execute:=TRUE , 
		Position:=setPosPosition , 
		Mode:= , 
		Options:= setPosOptions, 
		Done=> , 
		Busy=> , 
		Error=> , 
		ErrorID=> );
	IF mcSetPos.Done THEN//mcSetPos.Done信号只保持一个扫描周期
		setPosStep:=5000;//done
	ELSIF mcSetPos.Error OR mcSetPos.ErrorID<>0 THEN
		errorStep:=11;
		setPosStep:=10000;//error
	END_IF

	IF axisStopFlag OR NOT powerReady OR 0<>stopStep THEN
		setPosStep:=4000;//stop
	END_IF

4000://Stop
	mcSetPos(
		Axis:=axis , 
		Execute:=FALSE ,);
	setPosExecute:=FALSE;
	setPosBusy:=FALSE;
	setPosDone:=FALSE;
	setPosErrorDone:=FALSE;
	setPosStep:=0;
5000://Done
	mcSetPos(
		Axis:=axis , 
		Execute:=FALSE ,);
	setPosExecute:=FALSE;
	setPosBusy:=FALSE;
	setPosDone:=TRUE;
	setPosErrorDone:=FALSE;
	setPosStep:=0;
10000://Error
	mcSetPos(
		Axis:=axis , 
		Execute:=FALSE ,);
	setPosExecute:=FALSE;
	setPosBusy:=FALSE;
	setPosDone:=FALSE;
	setPosErrorDone:=TRUE;
	setPosStep:=0;
END_CASE
END_ACTION

//设定相对定位运行模式的距离和速度
METHOD setRel
VAR_INPUT
	dis:LREAL;//相对目标设定
	vel:LREAL;//速度设定
END_VAR
relDistance:=dis;
relVelocity:=vel;
END_METHOD

//设定速度运行模式的方向和速度
METHOD setVel
VAR_INPUT
	dire:BOOL;//方向设定, TRUE为正方向, FALSE为负方向
	vel:LREAL;//速度设定
END_VAR
velDirection:=dire;
velVelocity:=vel;
END_METHOD

ACTION Stop_ACT:
//轴停止函数--stopExecute触发条件是复归型

mcStop(
	Axis:=axis , 
	Execute:=, 
	Deceleration:= , 
	Jerk:= ,
	Options:= ,
	Done=>,
	Busy=> ,
	Active=> ,
	CommandAborted=> ,
	Error=> , 
	ErrorID=> );
	(*IF stopStep<>0 THEN
		stopStep:=0;
		stopErrorDone:=mcStop.Execute;
	END_IF*)
(*mcHalt(
	Axis:= axis, 
	Execute:= , 
	Deceleration:= , 
	Jerk:= , 
	BufferMode:= , 
	Options:= , 
	Done=> , 
	Busy=> , 
	Active=> , 
	CommandAborted=> , 
	Error=> , 
	ErrorID=> );*)
//(*
CASE stopStep OF
0:
	stopBusy:=FALSE;
	IF stopExecute AND powerReady (*AND bE_Stop*) THEN
		stopBusy:=TRUE;
		stopDone:=FALSE;
		stopErrorDone:=FALSE;
		stopStep:=10;
	END_IF
	stopExecute:=FALSE;
10:
	stopTimeout(IN:=FALSE);
	mcStop(
		Axis:=axis , 
		Execute:=FALSE,);
	(*mcHalt(
		Axis:=axis , 
		Execute:=FALSE,);*)
	stopStep:=20;
20:
	mcStop.Execute:=TRUE;
	mcStop.Deceleration:=stopDeceleration;
	mcStop.Jerk:=stopJerk;
	stopStep:=30;
30:
	//stopExecute:=FALSE;
	(*
	mcStop(
		Axis:=axis , 
		Execute:=TRUE, 
		Deceleration:=stopDeceleration , 
		Jerk:=stopJerk ,
		Options:= ,
		Done=>,
		Busy=> ,
		Active=> ,
		CommandAborted=> ,
		Error=> , 
		ErrorID=> );
	//*)
	(*
	mcHalt(
		Axis:= axis, 
		Execute:= TRUE, 
		Deceleration:= stopDeceleration, 
		Jerk:= , 
		BufferMode:= , 
		Options:= , 
		Done=> , 
		Busy=> , 
		Active=> , 
		CommandAborted=> , 
		Error=> , 
		ErrorID=> );
	//*)
	stopTimeout(IN:=NOT stopTimeout.Q,PT:=T#60S);
	
	IF mcStop.Done(* OR mcHalt.Done *) AND (axis.Status.NotMoving (*AND axis.Status.StandStill*)) THEN//mcStop.Done信号只保持一个扫描周期
		(*mcStop(
			Axis:=axis , 
			Execute:=FALSE, 
			Deceleration:=stopDeceleration , 
			Jerk:=stopJerk ,
			Options:= ,
			Done=>,
			Busy=> ,
			Active=> ,
			CommandAborted=> ,
			Error=> , 
			ErrorID=> );*)
		mcStop.Execute:=FALSE;
		(*mcHalt(
			Axis:=axis , 
			Execute:=FALSE,);*)
		stopStep:=40;
	ELSIF mcStop.Error OR mcStop.ErrorID<>0 (*OR mcHalt.Error OR mcHalt.ErrorID<>0*) THEN
		errorStep:=12;
		stopStep:=10000;//error
	ELSIF stopTimeout.Q THEN
		stopStep:=10;
	END_IF
40:
	mcReset(
		Axis:= axis, 
		Execute:= TRUE,
		Done=> , 
		Busy=> , 
		Error=> , 
		ErrorID=> );
	stopStep:=41;
41:
	stopStep:=5000;//done
	mcReset(
		Axis:= axis, 
		Execute:= FALSE,
		Done=> , 
		Busy=> , 
		Error=> , 
		ErrorID=> );

4000://Stop
	mcStop(
		Axis:=axis , 
		Execute:=FALSE ,);
	stopExecute:=FALSE;
	pauseExecute:=FALSE;
	stopBusy:=FALSE;
	stopDone:=FALSE;
	stopErrorDone:=FALSE;
	stopStep:=0;
5000://Done
	mcStop(
		Axis:=axis , 
		Execute:=FALSE ,);
	stopExecute:=FALSE;
	pauseExecute:=FALSE;
	stopBusy:=FALSE;
	stopDone:=TRUE;
	stopErrorDone:=FALSE;
	stopStep:=0;
	//homestep:=0;
10000://Error
	mcStop(
		Axis:=axis , 
		Execute:=FALSE ,);
	stopExecute:=FALSE;
	pauseExecute:=FALSE;
	stopBusy:=FALSE;
	stopDone:=FALSE;
	stopErrorDone:=TRUE;
	stopStep:=0;
END_CASE
//*)
END_ACTION

ACTION VelMove_ACT:
//轴的速度模式运行控制--velExecute触发条件是切换型
IF NOT bE_Stop THEN
	velStep:=0;
	velExecute:=FALSE;
END_IF
velCondition:=(NOT axisError AND NOT axisStopFlag 
				AND (NOT axisBusy OR homeBusy) 
				AND powerReady AND velConditionOuter 
				AND bE_Stop AND NOT axisPause);
mcVel(
	Axis:=axis , 
	Execute:= , 
	Velocity:= , 
	Acceleration:= , 
	Deceleration:= , 
	Jerk:= , 
	Direction:= , 
	BufferMode:= Tc2_MC2.MC_BufferMode.MC_Aborting, 
	Options:= , 
	InVelocity=> , 
	Busy=> , 
	Active=> , 
	CommandAborted=> , 
	Error=> , 
	ErrorID=>);
CASE velStep OF
0:
	velBusy:=FALSE;
	IF velExecute AND (NOT velCondition OR NOT powerEnable_Negative OR NOT powerEnable_Positive) THEN
		note_abs:=FALSE;
		note_jog:=FALSE;
		note_vel:=TRUE;
		note_home:=FALSE;
		note_rel:=FALSE;
	END_IF
	IF velExecute AND velCondition THEN
		note_abs:=FALSE;
		note_jog:=FALSE;
		note_vel:=FALSE;
		note_home:=FALSE;
		note_rel:=FALSE;
		velBusy:=TRUE;
		velDone:=FALSE;
		velErrorDone:=FALSE;
		velStep:=10;
		mcReset(
				Axis:= axis, 
				Execute:= TRUE,
				Done=> , 
				Busy=> , 
				Error=> , 
				ErrorID=> );
	ELSE
		velExecute:=FALSE;
	END_IF
	mcVel(
		Axis:=axis , 
		Execute:=FALSE);
	velChangeVel:=FALSE;
10:
	IF NOT axisStopFlag AND powerReady AND 0=stopStep THEN
			velStep:=20;
			mcReset(//陈培华
				Axis:= axis, 
				Execute:= FALSE,
				Done=> , 
				Busy=> , 
				Error=> , 
				ErrorID=> );
	END_IF
20:
	IF velDirection THEN
		IF (NOT bPLimitSwitch OR NOT bSoftPLimit OR NOT powerEnable_Positive) AND NOT homeBusy THEN
			axisStopFlag:=TRUE;
			
			IF NOT bPLimitSwitch THEN
				errorStep:=3;
			END_IF
			IF NOT bSoftPLimit THEN
				errorStep:=2;
			END_IF
			IF NOT powerEnable_Positive THEN
				errorStep:=19;
			END_IF
			velStep:=10000;//error
			RETURN;
		END_IF
	ELSE
		IF (NOT bNLimitSwitch OR NOT bSoftNLimit OR NOT powerEnable_Positive) AND NOT homeBusy THEN
			axisStopFlag:=TRUE;
			
			IF NOT bNLimitSwitch THEN
				errorStep:=4;
			END_IF
			IF NOT bSoftNLimit THEN
				errorStep:=2;
			END_IF
			IF NOT powerEnable_Positive THEN
				errorStep:=19;
			END_IF
			velStep:=10000;//error
			RETURN;
		END_IF
	END_IF
	IF velDirection THEN
		mcVel.Direction:=MC_Positive_Direction;
	ELSE
		mcVel.Direction:=MC_Negative_Direction;
	END_IF
	mcVel(
		Axis:=axis , 
		Execute:=TRUE , 
		Velocity:=velVelocity , 
		Acceleration:=velAcceleration , 
		Deceleration:=velDeceleration , 
		Jerk:=velJerk , 
		Direction:= , 
		BufferMode:= , 
		Options:= , 
		InVelocity=> , 
		Busy=> , 
		Active=> , 
		CommandAborted=> , 
		Error=> , 
		ErrorID=>);
	IF mcVel.Busy THEN
		velStep:=21;
	END_IF
21:
	(*mcVel(
		Axis:=axis , 
		Execute:=TRUE , 
		);*)
		velStep:=30;
30:
	IF velDirection THEN
		IF (NOT bPLimitSwitch OR NOT bSoftPLimit OR NOT powerEnable_Positive) AND NOT homeBusy THEN
			axisStopFlag:=TRUE;
			
			IF NOT bPLimitSwitch THEN
				errorStep:=3;
			END_IF
			IF NOT bSoftPLimit THEN
				errorStep:=2;
			END_IF
			IF NOT powerEnable_Positive THEN
				errorStep:=19;
			END_IF
			velStep:=10000;//error
			RETURN;
		END_IF
	ELSE
		IF (NOT bNLimitSwitch OR NOT bSoftNLimit OR NOT powerEnable_Positive) AND NOT homeBusy THEN
			axisStopFlag:=TRUE;
			
			IF NOT bNLimitSwitch THEN
				errorStep:=4;
			END_IF
			IF NOT bSoftNLimit THEN
				errorStep:=2;
			END_IF
			IF NOT powerEnable_Positive THEN
				errorStep:=19;
			END_IF
			velStep:=10000;//error
			RETURN;
		END_IF
	END_IF
	
	IF velChangeVel THEN
		velChangeVel:=FALSE;
	mcVel(
		Axis:=axis , 
		Execute:=FALSE , 
		);
		mcVel(
			Axis:=axis , 
			Execute:=TRUE , 
			Velocity:=velVelocity , 
			Acceleration:=velAcceleration , 
			Deceleration:=velDeceleration , 
			Jerk:=velJerk , 
			Direction:= , 
			BufferMode:= , 
			Options:= , 
			InVelocity=> , 
			Busy=> , 
			Active=> , 
			CommandAborted=> , 
			Error=> , 
			ErrorID=>);
	END_IF
	IF NOT velExecute THEN
		mcVel(
			Axis:=axis , 
			Execute:=FALSE ,);
		stopExecute:=TRUE;//轴停止
		velStep:=40;
	END_IF
	IF mcVel.Error OR mcVel.ErrorID<>0 THEN
		errorStep:=13;
		velStep:=10000;//error
	END_IF

	IF axisStopFlag OR NOT powerReady OR 0<>stopStep THEN
		velStep:=4000;//stop
	END_IF
	
40:
	velExecute:=FALSE;
	IF 0=stopStep THEN
		velStep:=5000;//done
	END_IF
4000://Stop
	mcVel(
		Axis:=axis , 
		Execute:=FALSE ,);
	velExecute:=FALSE;
	velBusy:=FALSE;
	velDone:=FALSE;
	velErrorDone:=FALSE;
	velStep:=0;
5000://Done
	mcVel(
		Axis:=axis , 
		Execute:=FALSE ,);
	velExecute:=FALSE;
	velBusy:=FALSE;
	velDone:=TRUE;
	velErrorDone:=FALSE;
	velStep:=0;
10000://Error
	mcVel(
		Axis:=axis , 
		Execute:=FALSE ,);
	velExecute:=FALSE;
	velBusy:=FALSE;
	velDone:=FALSE;
	velErrorDone:=TRUE;
	velStep:=0;
END_CASE
END_ACTION

ACTION VersionLog:
(*
旧版本: V1.0.0.0
(--------------------------------------------------)
新版本: V1.0.0.1
更新说明:
	1. 增加绝对运动三段变速触发功能
	2. 优化部分代码
(--------------------------------------------------)
新版本: V1.0.0.2
更新时间: 2019/09/16 8:30
更新说明:
	1. 修复轴停止在一直触发的情况下导致轴停止失效的bug
	2. 增加速度模式运行时动态变速触发功能
	3. 增加HMI按钮条件判断功能
	4. 优化部分代码
(--------------------------------------------------)
新版本: V1.0.0.3
更新时间: 2019/09/24 9:35
更新说明:
	1. 优化绝对运动的三段变速运动为可变多段变速
	2. 优化部分代码
(--------------------------------------------------)
新版本: V1.0.0.4
更新时间: 2019/10/10 18:55
更新说明:
	1. 增加 AXIS_REF 指针对象输出
(--------------------------------------------------)
新版本: V1.0.0.5
更新时间: 2019/11/04 8:55
更新说明:
	1. 修正驱动器回原点使能失败的bug
(--------------------------------------------------)
新版本: V1.0.0.6
更新时间: 2019/11/12 19:02
更新说明:
	1. 修改ABS运动变速位置不准问题
(--------------------------------------------------)
新版本: V1.0.1.0
更新时间: 2019/11/20 18:40
更新说明:
	1. 优化编写方式，减少扫描周期损耗
	2. 修改错误编码起始位，现改为从1开始
(--------------------------------------------------)
新版本: V1.0.1.1
更新时间: 2019/12/02
更新说明:
	1. 优化正负限位功能
	2. 增加正负软限位功能
(--------------------------------------------------)
新版本: V1.0.1.2
更新时间: 2020/03/23
更新说明:
	1. 优化报错功能
(--------------------------------------------------)
新版本: V1.0.1.3
更新时间: 2020/03/30
更新说明:
	1. 修正内部使能关闭后未及时开启导致无法使能的BUG
(--------------------------------------------------)
新版本: V1.0.1.4
更新时间: 2020/04/22
更新说明:
	1. 增加中文报警输出
(--------------------------------------------------)
新版本: V1.0.1.5
更新时间: 2020/09/12
更新说明:
	1. 处理ManualCtr_ACT下控制模式切换后可能导致掉使能的问题
(--------------------------------------------------)
新版本: V1.0.1.6
更新时间: 2020/09/16
更新说明:
	1. 开放错误ID、错误文本信息获取接口
(--------------------------------------------------)
新版本: V1.0.1.7
更新时间: 2020/10/06
更新说明:
	1. 移除控制模式变量，增加HMI启用条件
(--------------------------------------------------)
新版本: V1.0.1.8
更新时间: 2020/10/14
更新说明:
	1. 优化代码
(--------------------------------------------------)
新版本: V1.0.1.9
更新时间: 2020/11/4
更新说明:
	1. 处理轴停止控制步无法正常结束的bug
(--------------------------------------------------)
*)
END_ACTION

END_FUNCTION_BLOCK

// ---- POUs/BaseModule/ActionModule/cylinderModule/CylinderModule.TcPOU
(*
--报错编号0: 无报错
--报错编号1: Extend Error
--报错编号2: Retract Error
*)
FUNCTION_BLOCK CylinderModule
VAR_IN_OUT
	WarmHMI					:WARMStruct;
	NoteHMI					:NoteStruct;
	operatorLog				:printLogModule_EX;
END_VAR
VAR_INPUT
	HMIItf						:CylinderModuleHMI;//每个气缸对象都关联了一个HMI
	cylinderType				:CylinderType:=CylinderType_Default;//设置气缸的类型, 可通过该变量修改为真空发生器
	
	real_TimeMonitor			:BOOL:=TRUE;//实时状态检测
	extStep					    :UINT:=0;
	retStep					    :UINT:=0;
	extend						:BOOL:=FALSE;//伸出触发信号
	extCondition				:BOOL:=TRUE;//伸出启停条件
	retract						:BOOL:=FALSE;//收回触发信号
	retCondition				:BOOL:=TRUE;//收回启停条件
	reset						:BOOL:=FALSE;//复位信号
	stop						:BOOL:=FALSE;//停止信号
	power						:BOOL:=TRUE;//气缸动作后是否关闭继电器得电状态, TRUE--保持得电,FALSE--断开得电
	enable						:BOOL:=TRUE;//气缸禁用条件
	//ctrlMode					:ControlMode:=ControlMode.eManualCtrMode;//eManualCtrMode or eAutoCtrMode
	hmiEN						:BOOL:=TRUE;//HMI 启用条件
	
	errorDelayTime				:TIME:=T#3000MS;//气缸感应器感应超时
	//doneDelayTimeShort		:TIME:=T#100MS;//气缸感应到位延时---取消使用
	//doneDelayTimeLong			:TIME:=T#500MS;//无气缸感应到位延时---取消使用
	doneDelayTimeShortExtend	:TIME:=T#100MS;//气缸感应到位延时_伸出
	doneDelayTimeShortRetract	:TIME:=T#100MS;//气缸感应到位延时_收回
	doneDelayTimeLongExtend		:TIME:=T#500MS;//无气缸感应到位延时_伸出
	doneDelayTimeLongRetract	:TIME:=T#500MS;//无气缸感应到位延时_收回
	errorID						:UDINT:=0;//气缸错误报警分配的起始ID
	nameTXT						:STRING(255):='';//气缸名字
	inVacu						:REAL;
	viewForlineVac			:REAL:=100000;
	
